LIN {X 0,Y 467.559,Z 348.243,A -85,B 0,C 180,E1 -7440.293,E2 -7440.293} C_VEL
LIN {X 0,Y 467.621,Z 348.236,A -85,B 0,C 180,E1 -7443.199,E2 -7443.199} C_VEL
LIN {X 0,Y 467.597,Z 348.241,A -85,B 0,C 180,E1 -7446.467,E2 -7446.467} C_VEL
LIN {X 0,Y 467.627,Z 348.233,A -85,B 0,C 180,E1 -7449.776,E2 -7449.776} C_VEL
LIN {X 0,Y 467.613,Z 348.24,A -85,B 0,C 180,E1 -7452.506,E2 -7452.506} C_VEL
LIN {X 0,Y 467.61,Z 348.237,A -85,B 0,C 180,E1 -7455.196,E2 -7455.196} C_VEL
LIN {X 0,Y 467.659,Z 348.229,A -85,B 0,C 180,E1 -7457.854,E2 -7457.854} C_VEL
LIN {X 0,Y 467.685,Z 348.227,A -85,B 0,C 180,E1 -7461.356,E2 -7461.356} C_VEL
LIN {X 0,Y 467.738,Z 348.22,A -85,B 0,C 180,E1 -7463.962,E2 -7463.962} C_VEL
LIN {X 0,Y 467.863,Z 348.204,A -85,B 0,C 180,E1 -7467.416,E2 -7467.416} C_VEL
LIN {X 0,Y 467.885,Z 348.203,A -85,B 0,C 180,E1 -7469.999,E2 -7469.999} C_VEL
LIN {X 0,Y 467.862,Z 348.207,A -85,B 0,C 180,E1 -7472.582,E2 -7472.582} C_VEL
LIN {X 0,Y 467.747,Z 348.221,A -85,B 0,C 180,E1 -7476.036,E2 -7476.036} C_VEL
LIN {X 0,Y 467.683,Z 348.229,A -85,B 0,C 180,E1 -7478.642,E2 -7478.642} C_VEL
LIN {X 0,Y 467.656,Z 348.234,A -85,B 0,C 180,E1 -7482.144,E2 -7482.144} C_VEL
LIN {X 0,Y 467.666,Z 348.23,A -85,B 0,C 180,E1 -7485.892,E2 -7485.892} C_VEL
LIN {X 0,Y 467.623,Z 348.233,A -85,B 0,C 180,E1 -7489.307,E2 -7489.307} C_VEL
LIN {X 0,Y 467.534,Z 348.249,A -85,B 0,C 180,E1 -7492.073,E2 -7492.073} C_VEL
LIN {X 0,Y 467.601,Z 348.237,A -85,B 0,C 180,E1 -7494.886,E2 -7494.886} C_VEL
LIN {X 0,Y 467.625,Z 348.235,A -85,B 0,C 180,E1 -7497.767,E2 -7497.767} C_VEL
LIN {X 0,Y 467.569,Z 348.24,A -85,B 0,C 180,E1 -7501.045,E2 -7501.045} C_VEL
LIN {X 0,Y 467.586,Z 348.242,A -85,B 0,C 180,E1 -7504.242,E2 -7504.242} C_VEL
LIN {X 0,Y 467.547,Z 348.242,A -85,B 0,C 180,E1 -7507.186,E2 -7507.186} C_VEL
LIN {X 0,Y 467.596,Z 348.24,A -85,B 0,C 180,E1 -7510.261,E2 -7510.261} C_VEL
LIN {X 0,Y 467.613,Z 348.235,A -85,B 0,C 180,E1 -7512.57,E2 -7512.57} C_VEL
LIN {X 0,Y 467.568,Z 348.243,A -85,B 0,C 180,E1 -7516.175,E2 -7516.175} C_VEL
LIN {X 0,Y 467.584,Z 348.238,A -85,B 0,C 180,E1 -7518.72,E2 -7518.72} C_VEL
LIN {X 0,Y 467.572,Z 348.24,A -85,B 0,C 180,E1 -7521.405,E2 -7521.405} C_VEL
LIN {X 0,Y 467.555,Z 348.243,A -85,B 0,C 180,E1 -7524.259,E2 -7524.259} C_VEL
LIN {X 0,Y 467.574,Z 348.24,A -85,B 0,C 180,E1 -7527.32,E2 -7527.32} C_VEL
LIN {X 0,Y 467.569,Z 348.239,A -85,B 0,C 180,E1 -7530.665,E2 -7530.665} C_VEL
LIN {X 0,Y 467.619,Z 348.234,A -85,B 0,C 180,E1 -7533.2,E2 -7533.2} C_VEL
LIN {X 0,Y 467.583,Z 348.238,A -85,B 0,C 180,E1 -7536.467,E2 -7536.467} C_VEL
LIN {X 0,Y 467.614,Z 348.24,A -85,B 0,C 180,E1 -7539.777,E2 -7539.777} C_VEL
LIN {X 0,Y 467.6,Z 348.235,A -85,B 0,C 180,E1 -7542.506,E2 -7542.506} C_VEL
LIN {X 0,Y 467.597,Z 348.237,A -85,B 0,C 180,E1 -7545.196,E2 -7545.196} C_VEL
LIN {X 0,Y 467.673,Z 348.23,A -85,B 0,C 180,E1 -7547.855,E2 -7547.855} C_VEL
LIN {X 0,Y 467.673,Z 348.23,A -85,B 0,C 180,E1 -7551.357,E2 -7551.357} C_VEL
LIN {X 0,Y 467.734,Z 348.221,A -85,B 0,C 180,E1 -7553.963,E2 -7553.963} C_VEL
LIN {X 0,Y 467.851,Z 348.209,A -85,B 0,C 180,E1 -7557.417,E2 -7557.417} C_VEL
LIN {X 0,Y 467.873,Z 348.202,A -85,B 0,C 180,E1 -7560,E2 -7560} C_VEL
LIN {X 0,Y 467.852,Z 348.203,A -85,B 0,C 180,E1 -7562.583,E2 -7562.583} C_VEL
LIN {X 0,Y 467.742,Z 348.218,A -85,B 0,C 180,E1 -7566.038,E2 -7566.038} C_VEL
LIN {X 0,Y 467.673,Z 348.225,A -85,B 0,C 180,E1 -7568.643,E2 -7568.643} C_VEL
LIN {X 0,Y 467.682,Z 348.224,A -85,B 0,C 180,E1 -7572.379,E2 -7572.379} C_VEL
LIN {X 0,Y 467.64,Z 348.231,A -85,B 0,C 180,E1 -7575.886,E2 -7575.886} C_VEL
LIN {X 0,Y 467.615,Z 348.24,A -85,B 0,C 180,E1 -7579.308,E2 -7579.308} C_VEL
LIN {X 0,Y 467.528,Z 348.244,A -85,B 0,C 180,E1 -7582.074,E2 -7582.074} C_VEL
LIN {X 0,Y 467.595,Z 348.238,A -85,B 0,C 180,E1 -7584.888,E2 -7584.888} C_VEL
LIN {X 0,Y 467.619,Z 348.234,A -85,B 0,C 180,E1 -7587.769,E2 -7587.769} C_VEL
LIN {X 0,Y 467.561,Z 348.245,A -85,B 0,C 180,E1 -7591.046,E2 -7591.046} C_VEL
LIN {X 0,Y 467.582,Z 348.237,A -85,B 0,C 180,E1 -7594.244,E2 -7594.244} C_VEL
LIN {X 0,Y 467.546,Z 348.249,A -85,B 0,C 180,E1 -7597.188,E2 -7597.188} C_VEL
LIN {X 0,Y 467.592,Z 348.236,A -85,B 0,C 180,E1 -7600.263,E2 -7600.263} C_VEL
LIN {X 0,Y 467.613,Z 348.235,A -85,B 0,C 180,E1 -7602.572,E2 -7602.572} C_VEL
LIN {X 0,Y 467.569,Z 348.239,A -85,B 0,C 180,E1 -7606.177,E2 -7606.177} C_VEL
LIN {X 0,Y 467.585,Z 348.24,A -85,B 0,C 180,E1 -7608.723,E2 -7608.723} C_VEL
LIN {X 0,Y 467.575,Z 348.241,A -85,B 0,C 180,E1 -7611.408,E2 -7611.408} C_VEL
LIN {X 0,Y 467.56,Z 348.241,A -85,B 0,C 180,E1 -7614.261,E2 -7614.261} C_VEL
LIN {X 0,Y 467.579,Z 348.241,A -85,B 0,C 180,E1 -7617.322,E2 -7617.322} C_VEL
LIN {X 0,Y 467.577,Z 348.246,A -85,B 0,C 180,E1 -7620.666,E2 -7620.666} C_VEL
LIN {X 0,Y 467.629,Z 348.338,A -85,B 0,C 180,E1 -7621.989,E2 -7621.989} C_VEL
LIN {X 0,Y 470.457,Z 361.803,A -85,B 0,C 180,E1 -7624.329,E2 -7624.329} C_VEL
LIN {X 0,Y 470.48,Z 367.676,A -85,B 0,C 180,E1 -7625.276,E2 -7625.276} C_VEL
LIN {X 0,Y 469.476,Z 388.188,A -85,B 0,C 180,E1 -7628.508,E2 -7628.508} C_VEL
LIN {X 0,Y 468.653,Z 408.371,A -85,B 0,C 180,E1 -7631.645,E2 -7631.645} C_VEL
LIN {X 0,Y 468.38,Z 417.251,A -85,B 0,C 180,E1 -7633.015,E2 -7633.015} C_VEL
LIN {X 0,Y 470.991,Z 437.71,A -85,B 0,C 180,E1 -7633.47,E2 -7633.47} C_VEL
LIN {X 0,Y 470.045,Z 526.671,A -85,B 0,C 180,E1 -7634.999,E2 -7634.999} C_VEL
LIN {X 0,Y 469.641,Z 540.214,A -85,B 0,C 180,E1 -7635.402,E2 -7635.402} C_VEL
LIN {X 0,Y 469.224,Z 553.141,A -85,B 0,C 180,E1 -7635.97,E2 -7635.97} C_VEL
LIN {X 0,Y 468.755,Z 564.967,A -85,B 0,C 180,E1 -7636.674,E2 -7636.674} C_VEL
LIN {X 0,Y 468.309,Z 575.227,A -85,B 0,C 180,E1 -7637.443,E2 -7637.443} C_VEL
LIN {X 0,Y 467.916,Z 585.701,A -85,B 0,C 180,E1 -7638.412,E2 -7638.412} C_VEL
LIN {X 0,Y 467.556,Z 594.368,A -85,B 0,C 180,E1 -7639.39,E2 -7639.39} C_VEL
LIN {X 0,Y 467.25,Z 602.359,A -85,B 0,C 180,E1 -7640.478,E2 -7640.478} C_VEL
LIN {X 0,Y 466.998,Z 610.145,A -85,B 0,C 180,E1 -7641.781,E2 -7641.781} C_VEL
LIN {X 0,Y 466.858,Z 616.396,A -85,B 0,C 180,E1 -7643.084,E2 -7643.084} C_VEL
LIN {X 0,Y 466.797,Z 621.337,A -85,B 0,C 180,E1 -7644.385,E2 -7644.385} C_VEL
LIN {X 0,Y 466.717,Z 625.104,A -85,B 0,C 180,E1 -7645.683,E2 -7645.683} C_VEL
LIN {X 0,Y 466.77,Z 627.045,A -85,B 0,C 180,E1 -7646.548,E2 -7646.548} C_VEL
LIN {X 0,Y 466.778,Z 628.51,A -85,B 0,C 180,E1 -7647.412,E2 -7647.412} C_VEL
LIN {X 0,Y 466.698,Z 629.522,A -85,B 0,C 180,E1 -7648.275,E2 -7648.275} C_VEL
LIN {X 0,Y 466.637,Z 630.128,A -85,B 0,C 180,E1 -7649.138,E2 -7649.138} C_VEL
LIN {X 0,Y 466.631,Z 630.329,A -85,B 0,C 180,E1 -7650.001,E2 -7650.001} C_VEL
LIN {X 0,Y 466.639,Z 630.071,A -85,B 0,C 180,E1 -7650.864,E2 -7650.864} C_VEL
LIN {X 0,Y 466.7,Z 629.4,A -85,B 0,C 180,E1 -7651.727,E2 -7651.727} C_VEL
LIN {X 0,Y 466.8,Z 628.323,A -85,B 0,C 180,E1 -7652.59,E2 -7652.59} C_VEL
LIN {X 0,Y 466.784,Z 625.851,A -85,B 0,C 180,E1 -7653.886,E2 -7653.886} C_VEL
LIN {X 0,Y 466.78,Z 622.335,A -85,B 0,C 180,E1 -7655.184,E2 -7655.184} C_VEL
LIN {X 0,Y 466.88,Z 617.502,A -85,B 0,C 180,E1 -7656.532,E2 -7656.532} C_VEL
LIN {X 0,Y 466.986,Z 610.651,A -85,B 0,C 180,E1 -7658.003,E2 -7658.003} C_VEL
LIN {X 0,Y 467.174,Z 602.973,A -85,B 0,C 180,E1 -7659.308,E2 -7659.308} C_VEL
LIN {X 0,Y 467.499,Z 593.443,A -85,B 0,C 180,E1 -7660.613,E2 -7660.613} C_VEL
LIN {X 0,Y 467.83,Z 583.536,A -85,B 0,C 180,E1 -7661.702,E2 -7661.702} C_VEL
LIN {X 0,Y 468.246,Z 573.369,A -85,B 0,C 180,E1 -7662.615,E2 -7662.615} C_VEL
LIN {X 0,Y 468.759,Z 562.033,A -85,B 0,C 180,E1 -7663.439,E2 -7663.439} C_VEL
LIN {X 0,Y 469.19,Z 549.494,A -85,B 0,C 180,E1 -7664.144,E2 -7664.144} C_VEL
LIN {X 0,Y 469.678,Z 535.736,A -85,B 0,C 180,E1 -7664.71,E2 -7664.71} C_VEL
LIN {X 0,Y 470.109,Z 522.824,A -85,B 0,C 180,E1 -7665.056,E2 -7665.056} C_VEL
LIN {X 0,Y 471.009,Z 436.522,A -85,B 0,C 180,E1 -7666.593,E2 -7666.593} C_VEL
LIN {X 0,Y 468.235,Z 414.349,A -85,B 0,C 180,E1 -7667.146,E2 -7667.146} C_VEL
LIN {X 0,Y 468.975,Z 393.516,A -85,B 0,C 180,E1 -7670.392,E2 -7670.392} C_VEL
LIN {X 0,Y 469.735,Z 376.366,A -85,B 0,C 180,E1 -7673.126,E2 -7673.126} C_VEL
LIN {X 0,Y 470.441,Z 362.283,A -85,B 0,C 180,E1 -7675.437,E2 -7675.437} C_VEL
LIN {X 0,Y 468.39,Z 351.346,A -85,B 0,C 180,E1 -7677.457,E2 -7677.457} C_VEL
LIN {X 0,Y 467.622,Z 348.239,A -85,B 0,C 180,E1 -7678.074,E2 -7678.074} C_VEL
LIN {X 0,Y 467.588,Z 348.242,A -85,B 0,C 180,E1 -7681.741,E2 -7681.741} C_VEL
LIN {X 0,Y 467.571,Z 348.247,A -85,B 0,C 180,E1 -7684.833,E2 -7684.833} C_VEL
LIN {X 0,Y 467.571,Z 348.241,A -85,B 0,C 180,E1 -7688.045,E2 -7688.045} C_VEL
LIN {X 0,Y 467.583,Z 348.243,A -85,B 0,C 180,E1 -7691.277,E2 -7691.277} C_VEL
LIN {X 0,Y 467.559,Z 348.242,A -85,B 0,C 180,E1 -7693.821,E2 -7693.821} C_VEL
LIN {X 0,Y 467.562,Z 348.242,A -85,B 0,C 180,E1 -7696.256,E2 -7696.256} C_VEL
LIN {X 0,Y 467.584,Z 348.242,A -85,B 0,C 180,E1 -7698.723,E2 -7698.723} C_VEL
LIN {X 0,Y 467.57,Z 348.24,A -85,B 0,C 180,E1 -7701.956,E2 -7701.956} C_VEL
LIN {X 0,Y 467.569,Z 348.243,A -85,B 0,C 180,E1 -7705.168,E2 -7705.168} C_VEL
LIN {X 0,Y 467.588,Z 348.239,A -85,B 0,C 180,E1 -7708.26,E2 -7708.26} C_VEL
LIN {X 0,Y 467.582,Z 348.242,A -85,B 0,C 180,E1 -7711.251,E2 -7711.251} C_VEL
LIN {X 0,Y 467.616,Z 348.237,A -85,B 0,C 180,E1 -7714.16,E2 -7714.16} C_VEL
LIN {X 0,Y 467.582,Z 348.245,A -85,B 0,C 180,E1 -7716.996,E2 -7716.996} C_VEL
LIN {X 0,Y 467.628,Z 348.237,A -85,B 0,C 180,E1 -7719.777,E2 -7719.777} C_VEL
LIN {X 0,Y 467.655,Z 348.269,A -85,B 0,C 180,E1 -7721.415,E2 -7721.415} C_VEL
LIN {X 0,Y 468.732,Z 354.118,A -85,B 0,C 180,E1 -7722.999,E2 -7722.999} C_VEL
LIN {X 0,Y 471.442,Z 363.097,A -85,B 0,C 180,E1 -7723.298,E2 -7723.298} C_VEL
LIN {X 0,Y 471.589,Z 367.906,A -85,B 0,C 180,E1 -7723.398,E2 -7723.398} C_VEL
LIN {X 0,Y 470.308,Z 460.031,A -85,B 0,C 180,E1 -7725.09,E2 -7725.09} C_VEL
LIN {X 0,Y 470.102,Z 472.965,A -85,B 0,C 180,E1 -7725.498,E2 -7725.498} C_VEL
LIN {X 0,Y 469.752,Z 484.971,A -85,B 0,C 180,E1 -7726.04,E2 -7726.04} C_VEL
LIN {X 0,Y 469.45,Z 496.77,A -85,B 0,C 180,E1 -7726.758,E2 -7726.758} C_VEL
LIN {X 0,Y 468.982,Z 508.542,A -85,B 0,C 180,E1 -7727.67,E2 -7727.67} C_VEL
LIN {X 0,Y 468.613,Z 517.544,A -85,B 0,C 180,E1 -7728.538,E2 -7728.538} C_VEL
LIN {X 0,Y 468.237,Z 526.749,A -85,B 0,C 180,E1 -7729.623,E2 -7729.623} C_VEL
LIN {X 0,Y 467.818,Z 535.66,A -85,B 0,C 180,E1 -7730.924,E2 -7730.924} C_VEL
LIN {X 0,Y 467.483,Z 542.811,A -85,B 0,C 180,E1 -7732.224,E2 -7732.224} C_VEL
LIN {X 0,Y 467.173,Z 549.054,A -85,B 0,C 180,E1 -7733.679,E2 -7733.679} C_VEL
LIN {X 0,Y 467.075,Z 554.116,A -85,B 0,C 180,E1 -7735.253,E2 -7735.253} C_VEL
LIN {X 0,Y 467.009,Z 557.082,A -85,B 0,C 180,E1 -7736.549,E2 -7736.549} C_VEL
LIN {X 0,Y 466.845,Z 558.521,A -85,B 0,C 180,E1 -7737.411,E2 -7737.411} C_VEL
LIN {X 0,Y 466.667,Z 560.105,A -85,B 0,C 180,E1 -7739.137,E2 -7739.137} C_VEL
LIN {X 0,Y 466.655,Z 560.3,A -85,B 0,C 180,E1 -7740,E2 -7740} C_VEL
LIN {X 0,Y 466.664,Z 560.052,A -85,B 0,C 180,E1 -7740.863,E2 -7740.863} C_VEL
LIN {X 0,Y 466.841,Z 558.333,A -85,B 0,C 180,E1 -7742.588,E2 -7742.588} C_VEL
LIN {X 0,Y 466.975,Z 556.861,A -85,B 0,C 180,E1 -7743.451,E2 -7743.451} C_VEL
LIN {X 0,Y 467.019,Z 553.816,A -85,B 0,C 180,E1 -7744.748,E2 -7744.748} C_VEL
LIN {X 0,Y 467.166,Z 548.664,A -85,B 0,C 180,E1 -7746.318,E2 -7746.318} C_VEL
LIN {X 0,Y 467.356,Z 542.333,A -85,B 0,C 180,E1 -7747.778,E2 -7747.778} C_VEL
LIN {X 0,Y 467.699,Z 535.147,A -85,B 0,C 180,E1 -7749.078,E2 -7749.078} C_VEL
LIN {X 0,Y 468.076,Z 526.163,A -85,B 0,C 180,E1 -7750.38,E2 -7750.38} C_VEL
LIN {X 0,Y 468.481,Z 516.942,A -85,B 0,C 180,E1 -7751.465,E2 -7751.465} C_VEL
LIN {X 0,Y 468.95,Z 506.688,A -85,B 0,C 180,E1 -7752.441,E2 -7752.441} C_VEL
LIN {X 0,Y 469.25,Z 494.356,A -85,B 0,C 180,E1 -7753.379,E2 -7753.379} C_VEL
LIN {X 0,Y 469.629,Z 482.479,A -85,B 0,C 180,E1 -7754.074,E2 -7754.074} C_VEL
LIN {X 0,Y 470.016,Z 469.197,A -85,B 0,C 180,E1 -7754.643,E2 -7754.643} C_VEL
LIN {X 0,Y 470.283,Z 456.11,A -85,B 0,C 180,E1 -7755.022,E2 -7755.022} C_VEL
LIN {X 0,Y 471.084,Z 362.557,A -85,B 0,C 180,E1 -7756.634,E2 -7756.634} C_VEL
LIN {X 0,Y 467.987,Z 350.204,A -85,B 0,C 180,E1 -7756.984,E2 -7756.984} C_VEL
LIN {X 0,Y 467.63,Z 348.238,A -85,B 0,C 180,E1 -7757.492,E2 -7757.492} C_VEL
LIN {X 0,Y 467.627,Z 348.234,A -85,B 0,C 180,E1 -7760.223,E2 -7760.223} C_VEL
LIN {X 0,Y 467.574,Z 348.241,A -85,B 0,C 180,E1 -7763.943,E2 -7763.943} C_VEL
LIN {X 0,Y 467.62,Z 348.237,A -85,B 0,C 180,E1 -7766.8,E2 -7766.8} C_VEL
LIN {X 0,Y 467.559,Z 348.244,A -85,B 0,C 180,E1 -7769.738,E2 -7769.738} C_VEL
LIN {X 0,Y 467.588,Z 348.241,A -85,B 0,C 180,E1 -7772.758,E2 -7772.758} C_VEL
LIN {X 0,Y 467.558,Z 348.243,A -85,B 0,C 180,E1 -7775.889,E2 -7775.889} C_VEL
LIN {X 0,Y 467.587,Z 348.241,A -85,B 0,C 180,E1 -7779.144,E2 -7779.144} C_VEL
LIN {X 0,Y 467.591,Z 348.24,A -85,B 0,C 180,E1 -7782.567,E2 -7782.567} C_VEL
LIN {X 0,Y 467.575,Z 348.243,A -85,B 0,C 180,E1 -7785.053,E2 -7785.053} C_VEL
LIN {X 0,Y 467.593,Z 348.24,A -85,B 0,C 180,E1 -7787.439,E2 -7787.439} C_VEL
LIN {X 0,Y 467.587,Z 348.242,A -85,B 0,C 180,E1 -7790.855,E2 -7790.855} C_VEL
LIN {X 0,Y 467.564,Z 348.242,A -85,B 0,C 180,E1 -7794.26,E2 -7794.26} C_VEL
LIN {X 0,Y 467.586,Z 348.241,A -85,B 0,C 180,E1 -7797.32,E2 -7797.32} C_VEL
LIN {X 0,Y 467.559,Z 348.243,A -85,B 0,C 180,E1 -7800.293,E2 -7800.293} C_VEL
LIN {X 0,Y 466.907,Z 348.327,A -85,B 0,C 180,E1 -7801.013,E2 -7801.013} C_VEL
LIN {X 0,Y 464.063,Z 348.679,A -85,B 0,C 180,E1 -7802.182,E2 -7802.182} C_VEL
LIN {X 0,Y 461.661,Z 348.979,A -85,B 0,C 180,E1 -7803.125,E2 -7803.125} C_VEL
LIN {X 0,Y 460.643,Z 349.104,A -85,B 0,C 180,E1 -7803.854,E2 -7803.854} C_VEL
LIN {X 0,Y 460.568,Z 349.113,A -85,B 0,C 180,E1 -7804.1,E2 -7804.1} C_VEL
LIN {X 0,Y 460.55,Z 349.119,A -85,B 0,C 180,E1 -7806.623,E2 -7806.623} C_VEL
LIN {X 0,Y 460.555,Z 349.115,A -85,B 0,C 180,E1 -7809.452,E2 -7809.452} C_VEL
LIN {X 0,Y 460.563,Z 349.115,A -85,B 0,C 180,E1 -7812.229,E2 -7812.229} C_VEL
LIN {X 0,Y 460.569,Z 349.114,A -85,B 0,C 180,E1 -7814.964,E2 -7814.964} C_VEL
LIN {X 0,Y 460.615,Z 349.111,A -85,B 0,C 180,E1 -7818.558,E2 -7818.558} C_VEL
LIN {X 0,Y 460.698,Z 349.098,A -85,B 0,C 180,E1 -7822.108,E2 -7822.108} C_VEL
LIN {X 0,Y 460.697,Z 349.099,A -85,B 0,C 180,E1 -7824.747,E2 -7824.747} C_VEL
LIN {X 0,Y 460.828,Z 349.08,A -85,B 0,C 180,E1 -7827.377,E2 -7827.377} C_VEL
LIN {X 0,Y 460.856,Z 349.078,A -85,B 0,C 180,E1 -7829.999,E2 -7829.999} C_VEL
LIN {X 0,Y 460.827,Z 349.083,A -85,B 0,C 180,E1 -7832.621,E2 -7832.621} C_VEL
LIN {X 0,Y 460.713,Z 349.098,A -85,B 0,C 180,E1 -7836.129,E2 -7836.129} C_VEL
LIN {X 0,Y 460.63,Z 349.106,A -85,B 0,C 180,E1 -7838.775,E2 -7838.775} C_VEL
LIN {X 0,Y 460.613,Z 349.11,A -85,B 0,C 180,E1 -7842.444,E2 -7842.444} C_VEL
LIN {X 0,Y 460.621,Z 349.109,A -85,B 0,C 180,E1 -7846.006,E2 -7846.006} C_VEL
LIN {X 0,Y 460.568,Z 349.113,A -85,B 0,C 180,E1 -7849.614,E2 -7849.614} C_VEL
LIN {X 0,Y 460.51,Z 349.122,A -85,B 0,C 180,E1 -7852.427,E2 -7852.427} C_VEL
LIN {X 0,Y 460.566,Z 349.115,A -85,B 0,C 180,E1 -7855.801,E2 -7855.801} C_VEL
LIN {X 0,Y 460.556,Z 349.118,A -85,B 0,C 180,E1 -7858.231,E2 -7858.231} C_VEL
LIN {X 0,Y 460.521,Z 349.118,A -85,B 0,C 180,E1 -7861.283,E2 -7861.283} C_VEL
LIN {X 0,Y 460.53,Z 349.118,A -85,B 0,C 180,E1 -7864.505,E2 -7864.505} C_VEL
LIN {X 0,Y 460.526,Z 349.119,A -85,B 0,C 180,E1 -7867.619,E2 -7867.619} C_VEL
LIN {X 0,Y 460.558,Z 349.116,A -85,B 0,C 180,E1 -7870.272,E2 -7870.272} C_VEL
LIN {X 0,Y 460.518,Z 349.119,A -85,B 0,C 180,E1 -7873.371,E2 -7873.371} C_VEL
LIN {X 0,Y 460.518,Z 349.119,A -85,B 0,C 180,E1 -7876.627,E2 -7876.627} C_VEL
LIN {X 0,Y 460.557,Z 349.118,A -85,B 0,C 180,E1 -7879.726,E2 -7879.726} C_VEL
LIN {X 0,Y 460.521,Z 349.118,A -85,B 0,C 180,E1 -7882.518,E2 -7882.518} C_VEL
LIN {X 0,Y 460.541,Z 349.119,A -85,B 0,C 180,E1 -7885.623,E2 -7885.623} C_VEL
LIN {X 0,Y 460.528,Z 349.116,A -85,B 0,C 180,E1 -7888.744,E2 -7888.744} C_VEL
LIN {X 0,Y 460.55,Z 349.121,A -85,B 0,C 180,E1 -7891.767,E2 -7891.767} C_VEL
LIN {X 0,Y 460.55,Z 349.113,A -85,B 0,C 180,E1 -7894.705,E2 -7894.705} C_VEL
LIN {X 0,Y 460.503,Z 349.124,A -85,B 0,C 180,E1 -7897.571,E2 -7897.571} C_VEL
LIN {X 0,Y 460.56,Z 349.113,A -85,B 0,C 180,E1 -7900.384,E2 -7900.384} C_VEL
LIN {X 0,Y 460.621,Z 349.107,A -85,B 0,C 180,E1 -7904.06,E2 -7904.06} C_VEL
LIN {X 0,Y 460.62,Z 349.111,A -85,B 0,C 180,E1 -7907.666,E2 -7907.666} C_VEL
LIN {X 0,Y 460.62,Z 349.107,A -85,B 0,C 180,E1 -7911.224,E2 -7911.224} C_VEL
LIN {X 0,Y 460.7,Z 349.098,A -85,B 0,C 180,E1 -7913.87,E2 -7913.87} C_VEL
LIN {X 0,Y 460.816,Z 349.085,A -85,B 0,C 180,E1 -7917.378,E2 -7917.378} C_VEL
LIN {X 0,Y 460.844,Z 349.078,A -85,B 0,C 180,E1 -7920,E2 -7920} C_VEL
LIN {X 0,Y 460.817,Z 349.079,A -85,B 0,C 180,E1 -7922.623,E2 -7922.623} C_VEL
LIN {X 0,Y 460.707,Z 349.094,A -85,B 0,C 180,E1 -7926.13,E2 -7926.13} C_VEL
LIN {X 0,Y 460.62,Z 349.105,A -85,B 0,C 180,E1 -7928.776,E2 -7928.776} C_VEL
LIN {X 0,Y 460.624,Z 349.103,A -85,B 0,C 180,E1 -7932.457,E2 -7932.457} C_VEL
LIN {X 0,Y 460.59,Z 349.109,A -85,B 0,C 180,E1 -7935.998,E2 -7935.998} C_VEL
LIN {X 0,Y 460.562,Z 349.114,A -85,B 0,C 180,E1 -7938.903,E2 -7938.903} C_VEL
LIN {X 0,Y 460.507,Z 349.124,A -85,B 0,C 180,E1 -7941.486,E2 -7941.486} C_VEL
LIN {X 0,Y 460.534,Z 349.115,A -85,B 0,C 180,E1 -7944.333,E2 -7944.333} C_VEL
LIN {X 0,Y 460.576,Z 349.117,A -85,B 0,C 180,E1 -7947.244,E2 -7947.244} C_VEL
LIN {X 0,Y 460.503,Z 349.119,A -85,B 0,C 180,E1 -7950.241,E2 -7950.241} C_VEL
LIN {X 0,Y 460.522,Z 349.122,A -85,B 0,C 180,E1 -7953.326,E2 -7953.326} C_VEL
LIN {X 0,Y 460.473,Z 349.124,A -85,B 0,C 180,E1 -7956.53,E2 -7956.53} C_VEL
LIN {X 0,Y 460.572,Z 349.111,A -85,B 0,C 180,E1 -7959.858,E2 -7959.858} C_VEL
LIN {X 0,Y 460.537,Z 349.119,A -85,B 0,C 180,E1 -7962.905,E2 -7962.905} C_VEL
LIN {X 0,Y 460.519,Z 349.118,A -85,B 0,C 180,E1 -7965.83,E2 -7965.83} C_VEL
LIN {X 0,Y 460.538,Z 349.121,A -85,B 0,C 180,E1 -7968.991,E2 -7968.991} C_VEL
LIN {X 0,Y 460.544,Z 349.118,A -85,B 0,C 180,E1 -7971.27,E2 -7971.27} C_VEL
LIN {X 0,Y 460.511,Z 349.121,A -85,B 0,C 180,E1 -7974.556,E2 -7974.556} C_VEL
LIN {X 0,Y 460.531,Z 349.116,A -85,B 0,C 180,E1 -7977.717,E2 -7977.717} C_VEL
LIN {X 0,Y 460.547,Z 349.122,A -85,B 0,C 180,E1 -7980.771,E2 -7980.771} C_VEL
LIN {X 0,Y 460.615,Z 349.21,A -85,B 0,C 180,E1 -7981.773,E2 -7981.773} C_VEL
LIN {X 0,Y 463.432,Z 362.681,A -85,B 0,C 180,E1 -7984.153,E2 -7984.153} C_VEL
LIN {X 0,Y 463.587,Z 367.101,A -85,B 0,C 180,E1 -7984.883,E2 -7984.883} C_VEL
LIN {X 0,Y 462.657,Z 386.732,A -85,B 0,C 180,E1 -7988.027,E2 -7988.027} C_VEL
LIN {X 0,Y 461.713,Z 407.823,A -85,B 0,C 180,E1 -7991.359,E2 -7991.359} C_VEL
LIN {X 0,Y 461.379,Z 416.811,A -85,B 0,C 180,E1 -7992.767,E2 -7992.767} C_VEL
LIN {X 0,Y 464.125,Z 438.104,A -85,B 0,C 180,E1 -7993.252,E2 -7993.252} C_VEL
LIN {X 0,Y 463.091,Z 527.005,A -85,B 0,C 180,E1 -7994.825,E2 -7994.825} C_VEL
LIN {X 0,Y 462.662,Z 541.001,A -85,B 0,C 180,E1 -7995.261,E2 -7995.261} C_VEL
LIN {X 0,Y 462.254,Z 553.006,A -85,B 0,C 180,E1 -7995.81,E2 -7995.81} C_VEL
LIN {X 0,Y 461.726,Z 565.552,A -85,B 0,C 180,E1 -7996.579,E2 -7996.579} C_VEL
LIN {X 0,Y 461.276,Z 575.501,A -85,B 0,C 180,E1 -7997.35,E2 -7997.35} C_VEL
LIN {X 0,Y 460.852,Z 585.942,A -85,B 0,C 180,E1 -7998.344,E2 -7998.344} C_VEL
LIN {X 0,Y 460.44,Z 595.313,A -85,B 0,C 180,E1 -7999.447,E2 -7999.447} C_VEL
LIN {X 0,Y 460.096,Z 604.431,A -85,B 0,C 180,E1 -8000.772,E2 -8000.772} C_VEL
LIN {X 0,Y 459.87,Z 611.757,A -85,B 0,C 180,E1 -8002.095,E2 -8002.095} C_VEL
LIN {X 0,Y 459.771,Z 617.911,A -85,B 0,C 180,E1 -8003.507,E2 -8003.507} C_VEL
LIN {X 0,Y 459.71,Z 622.137,A -85,B 0,C 180,E1 -8004.738,E2 -8004.738} C_VEL
LIN {X 0,Y 459.625,Z 624.526,A -85,B 0,C 180,E1 -8005.616,E2 -8005.616} C_VEL
LIN {X 0,Y 459.699,Z 626.48,A -85,B 0,C 180,E1 -8006.495,E2 -8006.495} C_VEL
LIN {X 0,Y 459.692,Z 627.96,A -85,B 0,C 180,E1 -8007.372,E2 -8007.372} C_VEL
LIN {X 0,Y 459.637,Z 628.98,A -85,B 0,C 180,E1 -8008.249,E2 -8008.249} C_VEL
LIN {X 0,Y 459.569,Z 629.59,A -85,B 0,C 180,E1 -8009.125,E2 -8009.125} C_VEL
LIN {X 0,Y 459.56,Z 629.793,A -85,B 0,C 180,E1 -8010.001,E2 -8010.001} C_VEL
LIN {X 0,Y 459.571,Z 629.539,A -85,B 0,C 180,E1 -8010.877,E2 -8010.877} C_VEL
LIN {X 0,Y 459.639,Z 628.864,A -85,B 0,C 180,E1 -8011.753,E2 -8011.753} C_VEL
LIN {X 0,Y 459.714,Z 627.779,A -85,B 0,C 180,E1 -8012.63,E2 -8012.63} C_VEL
LIN {X 0,Y 459.695,Z 625.298,A -85,B 0,C 180,E1 -8013.946,E2 -8013.946} C_VEL
LIN {X 0,Y 459.714,Z 621.774,A -85,B 0,C 180,E1 -8015.264,E2 -8015.264} C_VEL
LIN {X 0,Y 459.803,Z 616.344,A -85,B 0,C 180,E1 -8016.778,E2 -8016.778} C_VEL
LIN {X 0,Y 459.911,Z 610.058,A -85,B 0,C 180,E1 -8018.127,E2 -8018.127} C_VEL
LIN {X 0,Y 460.12,Z 602.352,A -85,B 0,C 180,E1 -8019.452,E2 -8019.452} C_VEL
LIN {X 0,Y 460.467,Z 592.806,A -85,B 0,C 180,E1 -8020.777,E2 -8020.777} C_VEL
LIN {X 0,Y 460.852,Z 582.893,A -85,B 0,C 180,E1 -8021.882,E2 -8021.882} C_VEL
LIN {X 0,Y 461.298,Z 571.547,A -85,B 0,C 180,E1 -8022.907,E2 -8022.907} C_VEL
LIN {X 0,Y 461.875,Z 559.623,A -85,B 0,C 180,E1 -8023.755,E2 -8023.755} C_VEL
LIN {X 0,Y 462.404,Z 546.596,A -85,B 0,C 180,E1 -8024.468,E2 -8024.468} C_VEL
LIN {X 0,Y 462.861,Z 533.515,A -85,B 0,C 180,E1 -8024.988,E2 -8024.988} C_VEL
LIN {X 0,Y 463.297,Z 519.68,A -85,B 0,C 180,E1 -8025.339,E2 -8025.339} C_VEL
LIN {X 0,Y 464.308,Z 437.682,A -85,B 0,C 180,E1 -8026.84,E2 -8026.84} C_VEL
LIN {X 0,Y 461.277,Z 414.138,A -85,B 0,C 180,E1 -8027.441,E2 -8027.441} C_VEL
LIN {X 0,Y 461.24,Z 413.249,A -85,B 0,C 180,E1 -8027.524,E2 -8027.524} C_VEL
LIN {X 0,Y 462.007,Z 394.637,A -85,B 0,C 180,E1 -8030.48,E2 -8030.48} C_VEL
LIN {X 0,Y 462.878,Z 376.201,A -85,B 0,C 180,E1 -8033.489,E2 -8033.489} C_VEL
LIN {X 0,Y 463.607,Z 365.038,A -85,B 0,C 180,E1 -8035.358,E2 -8035.358} C_VEL
LIN {X 0,Y 462.855,Z 359.427,A -85,B 0,C 180,E1 -8036.381,E2 -8036.381} C_VEL
LIN {X 0,Y 460.579,Z 349.116,A -85,B 0,C 180,E1 -8038.418,E2 -8038.418} C_VEL
LIN {X 0,Y 460.526,Z 349.123,A -85,B 0,C 180,E1 -8041.284,E2 -8041.284} C_VEL
LIN {X 0,Y 460.538,Z 349.12,A -85,B 0,C 180,E1 -8044.506,E2 -8044.506} C_VEL
LIN {X 0,Y 460.507,Z 349.123,A -85,B 0,C 180,E1 -8047.624,E2 -8047.624} C_VEL
LIN {X 0,Y 460.547,Z 349.117,A -85,B 0,C 180,E1 -8050.27,E2 -8050.27} C_VEL
LIN {X 0,Y 460.506,Z 349.123,A -85,B 0,C 180,E1 -8053.376,E2 -8053.376} C_VEL
LIN {X 0,Y 460.506,Z 349.123,A -85,B 0,C 180,E1 -8056.625,E2 -8056.625} C_VEL
LIN {X 0,Y 460.547,Z 349.116,A -85,B 0,C 180,E1 -8059.731,E2 -8059.731} C_VEL
LIN {X 0,Y 460.505,Z 349.123,A -85,B 0,C 180,E1 -8062.524,E2 -8062.524} C_VEL
LIN {X 0,Y 460.551,Z 349.115,A -85,B 0,C 180,E1 -8065.624,E2 -8065.624} C_VEL
LIN {X 0,Y 460.543,Z 349.12,A -85,B 0,C 180,E1 -8068.745,E2 -8068.745} C_VEL
LIN {X 0,Y 460.587,Z 349.112,A -85,B 0,C 180,E1 -8072.254,E2 -8072.254} C_VEL
LIN {X 0,Y 460.564,Z 349.119,A -85,B 0,C 180,E1 -8074.706,E2 -8074.706} C_VEL
LIN {X 0,Y 460.516,Z 349.122,A -85,B 0,C 180,E1 -8077.571,E2 -8077.571} C_VEL
LIN {X 0,Y 460.58,Z 349.117,A -85,B 0,C 180,E1 -8080.8,E2 -8080.8} C_VEL
LIN {X 0,Y 460.596,Z 349.172,A -85,B 0,C 180,E1 -8081.091,E2 -8081.091} C_VEL
LIN {X 0,Y 461.661,Z 354.639,A -85,B 0,C 180,E1 -8082.66,E2 -8082.66} C_VEL
LIN {X 0,Y 464.627,Z 363.647,A -85,B 0,C 180,E1 -8082.998,E2 -8082.998} C_VEL
LIN {X 0,Y 464.969,Z 366.827,A -85,B 0,C 180,E1 -8083.079,E2 -8083.079} C_VEL
LIN {X 0,Y 463.503,Z 460.986,A -85,B 0,C 180,E1 -8084.865,E2 -8084.865} C_VEL
LIN {X 0,Y 463.269,Z 473.746,A -85,B 0,C 180,E1 -8085.279,E2 -8085.279} C_VEL
LIN {X 0,Y 462.915,Z 485.677,A -85,B 0,C 180,E1 -8085.829,E2 -8085.829} C_VEL
LIN {X 0,Y 462.569,Z 497.774,A -85,B 0,C 180,E1 -8086.58,E2 -8086.58} C_VEL
LIN {X 0,Y 462.078,Z 509.188,A -85,B 0,C 180,E1 -8087.482,E2 -8087.482} C_VEL
LIN {X 0,Y 461.684,Z 518.172,A -85,B 0,C 180,E1 -8088.364,E2 -8088.364} C_VEL
LIN {X 0,Y 461.282,Z 527.364,A -85,B 0,C 180,E1 -8089.465,E2 -8089.465} C_VEL
LIN {X 0,Y 460.839,Z 536.277,A -85,B 0,C 180,E1 -8090.785,E2 -8090.785} C_VEL
LIN {X 0,Y 460.495,Z 543.421,A -85,B 0,C 180,E1 -8092.105,E2 -8092.105} C_VEL
LIN {X 0,Y 460.194,Z 548.853,A -85,B 0,C 180,E1 -8093.363,E2 -8093.363} C_VEL
LIN {X 0,Y 460.125,Z 553.474,A -85,B 0,C 180,E1 -8094.742,E2 -8094.742} C_VEL
LIN {X 0,Y 459.979,Z 555.791,A -85,B 0,C 180,E1 -8095.619,E2 -8095.619} C_VEL
LIN {X 0,Y 459.963,Z 557.662,A -85,B 0,C 180,E1 -8096.496,E2 -8096.496} C_VEL
LIN {X 0,Y 459.794,Z 559.093,A -85,B 0,C 180,E1 -8097.372,E2 -8097.372} C_VEL
LIN {X 0,Y 459.659,Z 560.079,A -85,B 0,C 180,E1 -8098.248,E2 -8098.248} C_VEL
LIN {X 0,Y 459.598,Z 560.663,A -85,B 0,C 180,E1 -8099.124,E2 -8099.124} C_VEL
LIN {X 0,Y 459.583,Z 560.846,A -85,B 0,C 180,E1 -8100,E2 -8100} C_VEL
LIN {X 0,Y 459.595,Z 560.58,A -85,B 0,C 180,E1 -8100.876,E2 -8100.876} C_VEL
LIN {X 0,Y 459.789,Z 558.828,A -85,B 0,C 180,E1 -8102.628,E2 -8102.628} C_VEL
LIN {X 0,Y 459.899,Z 557.333,A -85,B 0,C 180,E1 -8103.504,E2 -8103.504} C_VEL
LIN {X 0,Y 459.966,Z 554.253,A -85,B 0,C 180,E1 -8104.821,E2 -8104.821} C_VEL
LIN {X 0,Y 460.057,Z 550.095,A -85,B 0,C 180,E1 -8106.139,E2 -8106.139} C_VEL
LIN {X 0,Y 460.27,Z 543.702,A -85,B 0,C 180,E1 -8107.678,E2 -8107.678} C_VEL
LIN {X 0,Y 460.612,Z 536.731,A -85,B 0,C 180,E1 -8108.998,E2 -8108.998} C_VEL
LIN {X 0,Y 460.937,Z 529.608,A -85,B 0,C 180,E1 -8110.099,E2 -8110.099} C_VEL
LIN {X 0,Y 461.303,Z 521.002,A -85,B 0,C 180,E1 -8111.201,E2 -8111.201} C_VEL
LIN {X 0,Y 461.809,Z 510.349,A -85,B 0,C 180,E1 -8112.302,E2 -8112.302} C_VEL
LIN {X 0,Y 462.19,Z 499.795,A -85,B 0,C 180,E1 -8113.184,E2 -8113.184} C_VEL
LIN {X 0,Y 462.568,Z 488.173,A -85,B 0,C 180,E1 -8113.957,E2 -8113.957} C_VEL
LIN {X 0,Y 462.944,Z 476.17,A -85,B 0,C 180,E1 -8114.563,E2 -8114.563} C_VEL
LIN {X 0,Y 463.216,Z 462.439,A -85,B 0,C 180,E1 -8115.06,E2 -8115.06} C_VEL
LIN {X 0,Y 463.402,Z 448.461,A -85,B 0,C 180,E1 -8115.363,E2 -8115.363} C_VEL
LIN {X 0,Y 464.387,Z 364.701,A -85,B 0,C 180,E1 -8116.825,E2 -8116.825} C_VEL
LIN {X 0,Y 461.858,Z 354.086,A -85,B 0,C 180,E1 -8117.109,E2 -8117.109} C_VEL
LIN {X 0,Y 460.859,Z 350.615,A -85,B 0,C 180,E1 -8117.235,E2 -8117.235} C_VEL
LIN {X 0,Y 460.6,Z 349.113,A -85,B 0,C 180,E1 -8117.654,E2 -8117.654} C_VEL
LIN {X 0,Y 460.556,Z 349.115,A -85,B 0,C 180,E1 -8120.547,E2 -8120.547} C_VEL
LIN {X 0,Y 460.539,Z 349.119,A -85,B 0,C 180,E1 -8123.704,E2 -8123.704} C_VEL
LIN {X 0,Y 460.563,Z 349.114,A -85,B 0,C 180,E1 -8126.265,E2 -8126.265} C_VEL
LIN {X 0,Y 460.545,Z 349.118,A -85,B 0,C 180,E1 -8129.231,E2 -8129.231} C_VEL
LIN {X 0,Y 460.536,Z 349.117,A -85,B 0,C 180,E1 -8132.284,E2 -8132.284} C_VEL
LIN {X 0,Y 460.515,Z 349.122,A -85,B 0,C 180,E1 -8135.445,E2 -8135.445} C_VEL
LIN {X 0,Y 460.549,Z 349.119,A -85,B 0,C 180,E1 -8138.897,E2 -8138.897} C_VEL
LIN {X 0,Y 460.527,Z 349.118,A -85,B 0,C 180,E1 -8142.181,E2 -8142.181} C_VEL
LIN {X 0,Y 460.521,Z 349.121,A -85,B 0,C 180,E1 -8145.411,E2 -8145.411} C_VEL
LIN {X 0,Y 460.536,Z 349.118,A -85,B 0,C 180,E1 -8148.397,E2 -8148.397} C_VEL
LIN {X 0,Y 460.531,Z 349.12,A -85,B 0,C 180,E1 -8151.266,E2 -8151.266} C_VEL
LIN {X 0,Y 460.515,Z 349.123,A -85,B 0,C 180,E1 -8154.554,E2 -8154.554} C_VEL
LIN {X 0,Y 460.535,Z 349.117,A -85,B 0,C 180,E1 -8157.715,E2 -8157.715} C_VEL
LIN {X 0,Y 460.544,Z 349.119,A -85,B 0,C 180,E1 -8160.768,E2 -8160.768} C_VEL
LIN {X 0,Y 460.567,Z 349.113,A -85,B 0,C 180,E1 -8163.734,E2 -8163.734} C_VEL
LIN {X 0,Y 460.568,Z 349.113,A -85,B 0,C 180,E1 -8164.1,E2 -8164.1} C_VEL
LIN {X 0,Y 459.912,Z 349.198,A -85,B 0,C 180,E1 -8164.83,E2 -8164.83} C_VEL
LIN {X 0,Y 457.023,Z 349.556,A -85,B 0,C 180,E1 -8166.014,E2 -8166.014} C_VEL
LIN {X 0,Y 454.579,Z 349.861,A -85,B 0,C 180,E1 -8166.969,E2 -8166.969} C_VEL
LIN {X 0,Y 453.545,Z 349.988,A -85,B 0,C 180,E1 -8167.708,E2 -8167.708} C_VEL
LIN {X 0,Y 453.47,Z 349.997,A -85,B 0,C 180,E1 -8167.958,E2 -8167.958} C_VEL
LIN {X 0,Y 453.526,Z 349.992,A -85,B 0,C 180,E1 -8171.008,E2 -8171.008} C_VEL
LIN {X 0,Y 453.572,Z 349.984,A -85,B 0,C 180,E1 -8173.879,E2 -8173.879} C_VEL
LIN {X 0,Y 453.566,Z 349.985,A -85,B 0,C 180,E1 -8177.47,E2 -8177.47} C_VEL
LIN {X 0,Y 453.595,Z 349.983,A -85,B 0,C 180,E1 -8181.086,E2 -8181.086} C_VEL
LIN {X 0,Y 453.672,Z 349.972,A -85,B 0,C 180,E1 -8183.774,E2 -8183.774} C_VEL
LIN {X 0,Y 453.768,Z 349.96,A -85,B 0,C 180,E1 -8187.336,E2 -8187.336} C_VEL
LIN {X 0,Y 453.826,Z 349.954,A -85,B 0,C 180,E1 -8189.999,E2 -8189.999} C_VEL
LIN {X 0,Y 453.767,Z 349.962,A -85,B 0,C 180,E1 -8192.662,E2 -8192.662} C_VEL
LIN {X 0,Y 453.68,Z 349.975,A -85,B 0,C 180,E1 -8196.224,E2 -8196.224} C_VEL
LIN {X 0,Y 453.593,Z 349.983,A -85,B 0,C 180,E1 -8198.912,E2 -8198.912} C_VEL
LIN {X 0,Y 453.563,Z 349.988,A -85,B 0,C 180,E1 -8202.528,E2 -8202.528} C_VEL
LIN {X 0,Y 453.556,Z 349.991,A -85,B 0,C 180,E1 -8206.194,E2 -8206.194} C_VEL
LIN {X 0,Y 453.519,Z 349.991,A -85,B 0,C 180,E1 -8209.04,E2 -8209.04} C_VEL
LIN {X 0,Y 453.475,Z 349.998,A -85,B 0,C 180,E1 -8211.835,E2 -8211.835} C_VEL
LIN {X 0,Y 453.512,Z 349.992,A -85,B 0,C 180,E1 -8214.733,E2 -8214.733} C_VEL
LIN {X 0,Y 453.536,Z 349.993,A -85,B 0,C 180,E1 -8217.96,E2 -8217.96} C_VEL
LIN {X 0,Y 453.48,Z 349.996,A -85,B 0,C 180,E1 -8220.758,E2 -8220.758} C_VEL
LIN {X 0,Y 453.474,Z 350,A -85,B 0,C 180,E1 -8223.911,E2 -8223.911} C_VEL
LIN {X 0,Y 453.467,Z 349.996,A -85,B 0,C 180,E1 -8227.187,E2 -8227.187} C_VEL
LIN {X 0,Y 453.531,Z 349.989,A -85,B 0,C 180,E1 -8229.444,E2 -8229.444} C_VEL
LIN {X 0,Y 453.485,Z 349.994,A -85,B 0,C 180,E1 -8232.99,E2 -8232.99} C_VEL
LIN {X 0,Y 453.47,Z 350.001,A -85,B 0,C 180,E1 -8235.78,E2 -8235.78} C_VEL
LIN {X 0,Y 453.49,Z 349.996,A -85,B 0,C 180,E1 -8238.211,E2 -8238.211} C_VEL
LIN {X 0,Y 453.528,Z 349.989,A -85,B 0,C 180,E1 -8240.786,E2 -8240.786} C_VEL
LIN {X 0,Y 453.45,Z 350.004,A -85,B 0,C 180,E1 -8243.917,E2 -8243.917} C_VEL
LIN {X 0,Y 453.475,Z 349.995,A -85,B 0,C 180,E1 -8247.151,E2 -8247.151} C_VEL
LIN {X 0,Y 453.505,Z 349.993,A -85,B 0,C 180,E1 -8250.271,E2 -8250.271} C_VEL
LIN {X 0,Y 453.505,Z 349.993,A -85,B 0,C 180,E1 -8253.294,E2 -8253.294} C_VEL
LIN {X 0,Y 453.494,Z 349.994,A -85,B 0,C 180,E1 -8256.238,E2 -8256.238} C_VEL
LIN {X 0,Y 453.473,Z 349.996,A -85,B 0,C 180,E1 -8259.117,E2 -8259.117} C_VEL
LIN {X 0,Y 453.503,Z 349.995,A -85,B 0,C 180,E1 -8261.944,E2 -8261.944} C_VEL
LIN {X 0,Y 453.54,Z 349.986,A -85,B 0,C 180,E1 -8264.726,E2 -8264.726} C_VEL
LIN {X 0,Y 453.592,Z 349.985,A -85,B 0,C 180,E1 -8267.472,E2 -8267.472} C_VEL
LIN {X 0,Y 453.584,Z 349.982,A -85,B 0,C 180,E1 -8271.087,E2 -8271.087} C_VEL
LIN {X 0,Y 453.668,Z 349.975,A -85,B 0,C 180,E1 -8273.775,E2 -8273.775} C_VEL
LIN {X 0,Y 453.757,Z 349.964,A -85,B 0,C 180,E1 -8277.337,E2 -8277.337} C_VEL
LIN {X 0,Y 453.815,Z 349.954,A -85,B 0,C 180,E1 -8280,E2 -8280} C_VEL
LIN {X 0,Y 453.757,Z 349.959,A -85,B 0,C 180,E1 -8282.663,E2 -8282.663} C_VEL
LIN {X 0,Y 453.673,Z 349.969,A -85,B 0,C 180,E1 -8286.225,E2 -8286.225} C_VEL
LIN {X 0,Y 453.584,Z 349.982,A -85,B 0,C 180,E1 -8288.914,E2 -8288.914} C_VEL
LIN {X 0,Y 453.592,Z 349.979,A -85,B 0,C 180,E1 -8292.551,E2 -8292.551} C_VEL
LIN {X 0,Y 453.535,Z 349.987,A -85,B 0,C 180,E1 -8296.196,E2 -8296.196} C_VEL
LIN {X 0,Y 453.512,Z 349.993,A -85,B 0,C 180,E1 -8299.042,E2 -8299.042} C_VEL
LIN {X 0,Y 453.468,Z 349.997,A -85,B 0,C 180,E1 -8301.837,E2 -8301.837} C_VEL
LIN {X 0,Y 453.506,Z 349.992,A -85,B 0,C 180,E1 -8304.735,E2 -8304.735} C_VEL
LIN {X 0,Y 453.529,Z 349.988,A -85,B 0,C 180,E1 -8307.962,E2 -8307.962} C_VEL
LIN {X 0,Y 453.459,Z 350,A -85,B 0,C 180,E1 -8311.526,E2 -8311.526} C_VEL
LIN {X 0,Y 453.482,Z 349.996,A -85,B 0,C 180,E1 -8314.779,E2 -8314.779} C_VEL
LIN {X 0,Y 453.479,Z 349.995,A -85,B 0,C 180,E1 -8318.31,E2 -8318.31} C_VEL
LIN {X 0,Y 453.51,Z 349.992,A -85,B 0,C 180,E1 -8320.607,E2 -8320.607} C_VEL
LIN {X 0,Y 453.477,Z 350,A -85,B 0,C 180,E1 -8323.249,E2 -8323.249} C_VEL
LIN {X 0,Y 453.472,Z 349.996,A -85,B 0,C 180,E1 -8325.782,E2 -8325.782} C_VEL
LIN {X 0,Y 453.491,Z 349.993,A -85,B 0,C 180,E1 -8328.212,E2 -8328.212} C_VEL
LIN {X 0,Y 453.529,Z 349.992,A -85,B 0,C 180,E1 -8330.788,E2 -8330.788} C_VEL
LIN {X 0,Y 453.455,Z 349.998,A -85,B 0,C 180,E1 -8333.919,E2 -8333.919} C_VEL
LIN {X 0,Y 453.48,Z 349.999,A -85,B 0,C 180,E1 -8337.153,E2 -8337.153} C_VEL
LIN {X 0,Y 453.512,Z 349.996,A -85,B 0,C 180,E1 -8340.272,E2 -8340.272} C_VEL
LIN {X 0,Y 453.544,Z 350.061,A -85,B 0,C 180,E1 -8341.552,E2 -8341.552} C_VEL
LIN {X 0,Y 456.643,Z 365.044,A -85,B 0,C 180,E1 -8344.23,E2 -8344.23} C_VEL
LIN {X 0,Y 456.222,Z 376.727,A -85,B 0,C 180,E1 -8346.149,E2 -8346.149} C_VEL
LIN {X 0,Y 455.258,Z 395.633,A -85,B 0,C 180,E1 -8349.204,E2 -8349.204} C_VEL
LIN {X 0,Y 454.384,Z 416.316,A -85,B 0,C 180,E1 -8352.505,E2 -8352.505} C_VEL
LIN {X 0,Y 457.254,Z 439.43,A -85,B 0,C 180,E1 -8353.053,E2 -8353.053} C_VEL
LIN {X 0,Y 456.197,Z 525.959,A -85,B 0,C 180,E1 -8354.618,E2 -8354.618} C_VEL
LIN {X 0,Y 455.74,Z 540.088,A -85,B 0,C 180,E1 -8355.06,E2 -8355.06} C_VEL
LIN {X 0,Y 455.266,Z 552.713,A -85,B 0,C 180,E1 -8355.644,E2 -8355.644} C_VEL
LIN {X 0,Y 454.765,Z 564.42,A -85,B 0,C 180,E1 -8356.37,E2 -8356.37} C_VEL
LIN {X 0,Y 454.243,Z 575.685,A -85,B 0,C 180,E1 -8357.255,E2 -8357.255} C_VEL
LIN {X 0,Y 453.771,Z 586.068,A -85,B 0,C 180,E1 -8358.272,E2 -8358.272} C_VEL
LIN {X 0,Y 453.309,Z 596.165,A -85,B 0,C 180,E1 -8359.505,E2 -8359.505} C_VEL
LIN {X 0,Y 453.001,Z 605.055,A -85,B 0,C 180,E1 -8360.851,E2 -8360.851} C_VEL
LIN {X 0,Y 452.76,Z 612.121,A -85,B 0,C 180,E1 -8362.195,E2 -8362.195} C_VEL
LIN {X 0,Y 452.632,Z 618.596,A -85,B 0,C 180,E1 -8363.761,E2 -8363.761} C_VEL
LIN {X 0,Y 452.571,Z 622.803,A -85,B 0,C 180,E1 -8365.101,E2 -8365.101} C_VEL
LIN {X 0,Y 452.63,Z 625.904,A -85,B 0,C 180,E1 -8366.44,E2 -8366.44} C_VEL
LIN {X 0,Y 452.611,Z 627.402,A -85,B 0,C 180,E1 -8367.331,E2 -8367.331} C_VEL
LIN {X 0,Y 452.577,Z 628.432,A -85,B 0,C 180,E1 -8368.221,E2 -8368.221} C_VEL
LIN {X 0,Y 452.504,Z 629.046,A -85,B 0,C 180,E1 -8369.111,E2 -8369.111} C_VEL
LIN {X 0,Y 452.492,Z 629.254,A -85,B 0,C 180,E1 -8370.001,E2 -8370.001} C_VEL
LIN {X 0,Y 452.506,Z 629.007,A -85,B 0,C 180,E1 -8370.891,E2 -8370.891} C_VEL
LIN {X 0,Y 452.579,Z 628.333,A -85,B 0,C 180,E1 -8371.781,E2 -8371.781} C_VEL
LIN {X 0,Y 452.632,Z 627.243,A -85,B 0,C 180,E1 -8372.671,E2 -8372.671} C_VEL
LIN {X 0,Y 452.609,Z 624.756,A -85,B 0,C 180,E1 -8374.008,E2 -8374.008} C_VEL
LIN {X 0,Y 452.625,Z 621.22,A -85,B 0,C 180,E1 -8375.347,E2 -8375.347} C_VEL
LIN {X 0,Y 452.712,Z 615.991,A -85,B 0,C 180,E1 -8376.833,E2 -8376.833} C_VEL
LIN {X 0,Y 452.832,Z 609.489,A -85,B 0,C 180,E1 -8378.255,E2 -8378.255} C_VEL
LIN {X 0,Y 453.063,Z 601.778,A -85,B 0,C 180,E1 -8379.6,E2 -8379.6} C_VEL
LIN {X 0,Y 453.454,Z 592.215,A -85,B 0,C 180,E1 -8380.946,E2 -8380.946} C_VEL
LIN {X 0,Y 453.796,Z 583.408,A -85,B 0,C 180,E1 -8381.956,E2 -8381.956} C_VEL
LIN {X 0,Y 454.268,Z 572.575,A -85,B 0,C 180,E1 -8382.973,E2 -8382.973} C_VEL
LIN {X 0,Y 454.876,Z 560.823,A -85,B 0,C 180,E1 -8383.857,E2 -8383.857} C_VEL
LIN {X 0,Y 455.414,Z 548.344,A -85,B 0,C 180,E1 -8384.581,E2 -8384.581} C_VEL
LIN {X 0,Y 455.941,Z 534.763,A -85,B 0,C 180,E1 -8385.164,E2 -8385.164} C_VEL
LIN {X 0,Y 456.45,Z 521.03,A -85,B 0,C 180,E1 -8385.547,E2 -8385.547} C_VEL
LIN {X 0,Y 457.527,Z 438.056,A -85,B 0,C 180,E1 -8387.12,E2 -8387.12} C_VEL
LIN {X 0,Y 454.672,Z 415.482,A -85,B 0,C 180,E1 -8387.719,E2 -8387.719} C_VEL
LIN {X 0,Y 454.293,Z 412.967,A -85,B 0,C 180,E1 -8387.793,E2 -8387.793} C_VEL
LIN {X 0,Y 455.11,Z 394.419,A -85,B 0,C 180,E1 -8390.805,E2 -8390.805} C_VEL
LIN {X 0,Y 456.116,Z 376.11,A -85,B 0,C 180,E1 -8393.859,E2 -8393.859} C_VEL
LIN {X 0,Y 456.753,Z 366.407,A -85,B 0,C 180,E1 -8395.521,E2 -8395.521} C_VEL
LIN {X 0,Y 455.751,Z 359.617,A -85,B 0,C 180,E1 -8396.812,E2 -8396.812} C_VEL
LIN {X 0,Y 453.507,Z 349.999,A -85,B 0,C 180,E1 -8398.808,E2 -8398.808} C_VEL
LIN {X 0,Y 453.47,Z 350.001,A -85,B 0,C 180,E1 -8401.8,E2 -8401.8} C_VEL
LIN {X 0,Y 453.486,Z 350.001,A -85,B 0,C 180,E1 -8404.99,E2 -8404.99} C_VEL
LIN {X 0,Y 453.47,Z 349.999,A -85,B 0,C 180,E1 -8408.312,E2 -8408.312} C_VEL
LIN {X 0,Y 453.499,Z 349.997,A -85,B 0,C 180,E1 -8410.609,E2 -8410.609} C_VEL
LIN {X 0,Y 453.461,Z 350.001,A -85,B 0,C 180,E1 -8413.245,E2 -8413.245} C_VEL
LIN {X 0,Y 453.472,Z 349.997,A -85,B 0,C 180,E1 -8415.779,E2 -8415.779} C_VEL
LIN {X 0,Y 453.485,Z 349.994,A -85,B 0,C 180,E1 -8418.21,E2 -8418.21} C_VEL
LIN {X 0,Y 453.515,Z 349.995,A -85,B 0,C 180,E1 -8420.791,E2 -8420.791} C_VEL
LIN {X 0,Y 453.459,Z 349.997,A -85,B 0,C 180,E1 -8423.917,E2 -8423.917} C_VEL
LIN {X 0,Y 453.488,Z 349.998,A -85,B 0,C 180,E1 -8427.151,E2 -8427.151} C_VEL
LIN {X 0,Y 453.48,Z 349.998,A -85,B 0,C 180,E1 -8430.269,E2 -8430.269} C_VEL
LIN {X 0,Y 453.512,Z 349.996,A -85,B 0,C 180,E1 -8433.294,E2 -8433.294} C_VEL
LIN {X 0,Y 453.508,Z 349.995,A -85,B 0,C 180,E1 -8436.239,E2 -8436.239} C_VEL
LIN {X 0,Y 453.488,Z 350,A -85,B 0,C 180,E1 -8439.118,E2 -8439.118} C_VEL
LIN {X 0,Y 453.563,Z 350.058,A -85,B 0,C 180,E1 -8440.734,E2 -8440.734} C_VEL
LIN {X 0,Y 454.656,Z 355.506,A -85,B 0,C 180,E1 -8442.329,E2 -8442.329} C_VEL
LIN {X 0,Y 458.208,Z 365.762,A -85,B 0,C 180,E1 -8442.732,E2 -8442.732} C_VEL
LIN {X 0,Y 457.192,Z 428.242,A -85,B 0,C 180,E1 -8443.965,E2 -8443.965} C_VEL
LIN {X 0,Y 456.728,Z 461.159,A -85,B 0,C 180,E1 -8444.607,E2 -8444.607} C_VEL
LIN {X 0,Y 456.457,Z 474.721,A -85,B 0,C 180,E1 -8445.055,E2 -8445.055} C_VEL
LIN {X 0,Y 456.087,Z 486.525,A -85,B 0,C 180,E1 -8445.613,E2 -8445.613} C_VEL
LIN {X 0,Y 455.717,Z 498.683,A -85,B 0,C 180,E1 -8446.385,E2 -8446.385} C_VEL
LIN {X 0,Y 455.186,Z 509.91,A -85,B 0,C 180,E1 -8447.29,E2 -8447.29} C_VEL
LIN {X 0,Y 454.764,Z 518.863,A -85,B 0,C 180,E1 -8448.184,E2 -8448.184} C_VEL
LIN {X 0,Y 454.357,Z 528.034,A -85,B 0,C 180,E1 -8449.303,E2 -8449.303} C_VEL
LIN {X 0,Y 453.869,Z 536.936,A -85,B 0,C 180,E1 -8450.643,E2 -8450.643} C_VEL
LIN {X 0,Y 453.51,Z 544.061,A -85,B 0,C 180,E1 -8451.983,E2 -8451.983} C_VEL
LIN {X 0,Y 453.158,Z 549.695,A -85,B 0,C 180,E1 -8453.319,E2 -8453.319} C_VEL
LIN {X 0,Y 453.093,Z 554.086,A -85,B 0,C 180,E1 -8454.66,E2 -8454.66} C_VEL
LIN {X 0,Y 452.935,Z 556.399,A -85,B 0,C 180,E1 -8455.55,E2 -8455.55} C_VEL
LIN {X 0,Y 452.919,Z 558.264,A -85,B 0,C 180,E1 -8456.441,E2 -8456.441} C_VEL
LIN {X 0,Y 452.745,Z 559.679,A -85,B 0,C 180,E1 -8457.331,E2 -8457.331} C_VEL
LIN {X 0,Y 452.6,Z 560.655,A -85,B 0,C 180,E1 -8458.22,E2 -8458.22} C_VEL
LIN {X 0,Y 452.531,Z 561.227,A -85,B 0,C 180,E1 -8459.11,E2 -8459.11} C_VEL
LIN {X 0,Y 452.514,Z 561.394,A -85,B 0,C 180,E1 -8460,E2 -8460} C_VEL
LIN {X 0,Y 452.528,Z 561.107,A -85,B 0,C 180,E1 -8460.89,E2 -8460.89} C_VEL
LIN {X 0,Y 452.595,Z 560.414,A -85,B 0,C 180,E1 -8461.78,E2 -8461.78} C_VEL
LIN {X 0,Y 452.738,Z 559.32,A -85,B 0,C 180,E1 -8462.669,E2 -8462.669} C_VEL
LIN {X 0,Y 452.828,Z 557.797,A -85,B 0,C 180,E1 -8463.559,E2 -8463.559} C_VEL
LIN {X 0,Y 452.912,Z 554.677,A -85,B 0,C 180,E1 -8464.896,E2 -8464.896} C_VEL
LIN {X 0,Y 453.025,Z 550.472,A -85,B 0,C 180,E1 -8466.234,E2 -8466.234} C_VEL
LIN {X 0,Y 453.256,Z 544.021,A -85,B 0,C 180,E1 -8467.798,E2 -8467.798} C_VEL
LIN {X 0,Y 453.606,Z 536.991,A -85,B 0,C 180,E1 -8469.138,E2 -8469.138} C_VEL
LIN {X 0,Y 453.996,Z 528.167,A -85,B 0,C 180,E1 -8470.48,E2 -8470.48} C_VEL
LIN {X 0,Y 454.469,Z 518.114,A -85,B 0,C 180,E1 -8471.71,E2 -8471.71} C_VEL
LIN {X 0,Y 454.983,Z 508.072,A -85,B 0,C 180,E1 -8472.7,E2 -8472.7} C_VEL
LIN {X 0,Y 455.293,Z 497.133,A -85,B 0,C 180,E1 -8473.572,E2 -8473.572} C_VEL
LIN {X 0,Y 455.724,Z 484.818,A -85,B 0,C 180,E1 -8474.342,E2 -8474.342} C_VEL
LIN {X 0,Y 456.154,Z 472.168,A -85,B 0,C 180,E1 -8474.927,E2 -8474.927} C_VEL
LIN {X 0,Y 456.422,Z 460.12,A -85,B 0,C 180,E1 -8475.318,E2 -8475.318} C_VEL
LIN {X 0,Y 456.622,Z 436.807,A -85,B 0,C 180,E1 -8475.769,E2 -8475.769} C_VEL
LIN {X 0,Y 457.41,Z 364.774,A -85,B 0,C 180,E1 -8477.068,E2 -8477.068} C_VEL
LIN {X 0,Y 454.618,Z 354.144,A -85,B 0,C 180,E1 -8477.368,E2 -8477.368} C_VEL
LIN {X 0,Y 453.743,Z 351.101,A -85,B 0,C 180,E1 -8477.468,E2 -8477.468} C_VEL
LIN {X 0,Y 453.548,Z 349.991,A -85,B 0,C 180,E1 -8477.763,E2 -8477.763} C_VEL
LIN {X 0,Y 453.487,Z 349.998,A -85,B 0,C 180,E1 -8480.882,E2 -8480.882} C_VEL
LIN {X 0,Y 453.502,Z 349.995,A -85,B 0,C 180,E1 -8483.887,E2 -8483.887} C_VEL
LIN {X 0,Y 453.509,Z 349.994,A -85,B 0,C 180,E1 -8486.706,E2 -8486.706} C_VEL
LIN {X 0,Y 453.477,Z 349.998,A -85,B 0,C 180,E1 -8489.784,E2 -8489.784} C_VEL
LIN {X 0,Y 453.495,Z 349.996,A -85,B 0,C 180,E1 -8493.189,E2 -8493.189} C_VEL
LIN {X 0,Y 453.457,Z 349.999,A -85,B 0,C 180,E1 -8496.299,E2 -8496.299} C_VEL
LIN {X 0,Y 453.51,Z 349.994,A -85,B 0,C 180,E1 -8499.448,E2 -8499.448} C_VEL
LIN {X 0,Y 453.468,Z 350,A -85,B 0,C 180,E1 -8502.994,E2 -8502.994} C_VEL
LIN {X 0,Y 453.47,Z 349.998,A -85,B 0,C 180,E1 -8505.779,E2 -8505.779} C_VEL
LIN {X 0,Y 453.483,Z 349.996,A -85,B 0,C 180,E1 -8508.209,E2 -8508.209} C_VEL
LIN {X 0,Y 453.514,Z 349.995,A -85,B 0,C 180,E1 -8510.79,E2 -8510.79} C_VEL
LIN {X 0,Y 453.459,Z 349.999,A -85,B 0,C 180,E1 -8513.917,E2 -8513.917} C_VEL
LIN {X 0,Y 453.487,Z 349.997,A -85,B 0,C 180,E1 -8517.151,E2 -8517.151} C_VEL
LIN {X 0,Y 453.479,Z 349.997,A -85,B 0,C 180,E1 -8520.268,E2 -8520.268} C_VEL
LIN {X 0,Y 453.511,Z 349.994,A -85,B 0,C 180,E1 -8523.293,E2 -8523.293} C_VEL
LIN {X 0,Y 453.508,Z 349.994,A -85,B 0,C 180,E1 -8526.238,E2 -8526.238} C_VEL
LIN {X 0,Y 453.47,Z 349.997,A -85,B 0,C 180,E1 -8527.958,E2 -8527.958} C_VEL
LIN {X 0,Y 452.831,Z 350.08,A -85,B 0,C 180,E1 -8528.699,E2 -8528.699} C_VEL
LIN {X 0,Y 449.998,Z 350.433,A -85,B 0,C 180,E1 -8529.904,E2 -8529.904} C_VEL
LIN {X 0,Y 447.582,Z 350.732,A -85,B 0,C 180,E1 -8530.875,E2 -8530.875} C_VEL
LIN {X 0,Y 446.539,Z 350.861,A -85,B 0,C 180,E1 -8531.626,E2 -8531.626} C_VEL
LIN {X 0,Y 446.451,Z 350.871,A -85,B 0,C 180,E1 -8531.88,E2 -8531.88} C_VEL
LIN {X 0,Y 446.511,Z 350.868,A -85,B 0,C 180,E1 -8534.479,E2 -8534.479} C_VEL
LIN {X 0,Y 446.521,Z 350.865,A -85,B 0,C 180,E1 -8538.192,E2 -8538.192} C_VEL
LIN {X 0,Y 446.603,Z 350.853,A -85,B 0,C 180,E1 -8541.857,E2 -8541.857} C_VEL
LIN {X 0,Y 446.645,Z 350.85,A -85,B 0,C 180,E1 -8544.582,E2 -8544.582} C_VEL
LIN {X 0,Y 446.712,Z 350.839,A -85,B 0,C 180,E1 -8547.294,E2 -8547.294} C_VEL
LIN {X 0,Y 446.796,Z 350.83,A -85,B 0,C 180,E1 -8549.999,E2 -8549.999} C_VEL
LIN {X 0,Y 446.711,Z 350.84,A -85,B 0,C 180,E1 -8552.704,E2 -8552.704} C_VEL
LIN {X 0,Y 446.649,Z 350.851,A -85,B 0,C 180,E1 -8556.323,E2 -8556.323} C_VEL
LIN {X 0,Y 446.539,Z 350.861,A -85,B 0,C 180,E1 -8559.054,E2 -8559.054} C_VEL
LIN {X 0,Y 446.521,Z 350.864,A -85,B 0,C 180,E1 -8562.729,E2 -8562.729} C_VEL
LIN {X 0,Y 446.518,Z 350.867,A -85,B 0,C 180,E1 -8566.237,E2 -8566.237} C_VEL
LIN {X 0,Y 446.468,Z 350.869,A -85,B 0,C 180,E1 -8569.302,E2 -8569.302} C_VEL
LIN {X 0,Y 446.417,Z 350.88,A -85,B 0,C 180,E1 -8572.198,E2 -8572.198} C_VEL
LIN {X 0,Y 446.456,Z 350.87,A -85,B 0,C 180,E1 -8575.151,E2 -8575.151} C_VEL
LIN {X 0,Y 446.481,Z 350.871,A -85,B 0,C 180,E1 -8578.177,E2 -8578.177} C_VEL
LIN {X 0,Y 446.416,Z 350.875,A -85,B 0,C 180,E1 -8581.299,E2 -8581.299} C_VEL
LIN {X 0,Y 446.426,Z 350.875,A -85,B 0,C 180,E1 -8584.522,E2 -8584.522} C_VEL
LIN {X 0,Y 446.434,Z 350.877,A -85,B 0,C 180,E1 -8588.082,E2 -8588.082} C_VEL
LIN {X 0,Y 446.442,Z 350.872,A -85,B 0,C 180,E1 -8590.92,E2 -8590.92} C_VEL
LIN {X 0,Y 446.439,Z 350.877,A -85,B 0,C 180,E1 -8593.839,E2 -8593.839} C_VEL
LIN {X 0,Y 446.44,Z 350.873,A -85,B 0,C 180,E1 -8596.396,E2 -8596.396} C_VEL
LIN {X 0,Y 446.463,Z 350.874,A -85,B 0,C 180,E1 -8599.804,E2 -8599.804} C_VEL
LIN {X 0,Y 446.427,Z 350.876,A -85,B 0,C 180,E1 -8602.123,E2 -8602.123} C_VEL
LIN {X 0,Y 446.423,Z 350.876,A -85,B 0,C 180,E1 -8605.476,E2 -8605.476} C_VEL
LIN {X 0,Y 446.411,Z 350.875,A -85,B 0,C 180,E1 -8608.699,E2 -8608.699} C_VEL
LIN {X 0,Y 446.475,Z 350.873,A -85,B 0,C 180,E1 -8611.821,E2 -8611.821} C_VEL
LIN {X 0,Y 446.449,Z 350.87,A -85,B 0,C 180,E1 -8614.847,E2 -8614.847} C_VEL
LIN {X 0,Y 446.439,Z 350.873,A -85,B 0,C 180,E1 -8618.244,E2 -8618.244} C_VEL
LIN {X 0,Y 446.449,Z 350.877,A -85,B 0,C 180,E1 -8621.649,E2 -8621.649} C_VEL
LIN {X 0,Y 446.506,Z 350.863,A -85,B 0,C 180,E1 -8624.48,E2 -8624.48} C_VEL
LIN {X 0,Y 446.53,Z 350.861,A -85,B 0,C 180,E1 -8628.193,E2 -8628.193} C_VEL
LIN {X 0,Y 446.59,Z 350.856,A -85,B 0,C 180,E1 -8631.858,E2 -8631.858} C_VEL
LIN {X 0,Y 446.637,Z 350.846,A -85,B 0,C 180,E1 -8634.583,E2 -8634.583} C_VEL
LIN {X 0,Y 446.701,Z 350.842,A -85,B 0,C 180,E1 -8637.295,E2 -8637.295} C_VEL
LIN {X 0,Y 446.785,Z 350.829,A -85,B 0,C 180,E1 -8640,E2 -8640} C_VEL
LIN {X 0,Y 446.701,Z 350.838,A -85,B 0,C 180,E1 -8642.705,E2 -8642.705} C_VEL
LIN {X 0,Y 446.642,Z 350.845,A -85,B 0,C 180,E1 -8646.324,E2 -8646.324} C_VEL
LIN {X 0,Y 446.53,Z 350.862,A -85,B 0,C 180,E1 -8649.056,E2 -8649.056} C_VEL
LIN {X 0,Y 446.525,Z 350.861,A -85,B 0,C 180,E1 -8652.73,E2 -8652.73} C_VEL
LIN {X 0,Y 446.481,Z 350.865,A -85,B 0,C 180,E1 -8656.46,E2 -8656.46} C_VEL
LIN {X 0,Y 446.46,Z 350.875,A -85,B 0,C 180,E1 -8659.304,E2 -8659.304} C_VEL
LIN {X 0,Y 446.409,Z 350.874,A -85,B 0,C 180,E1 -8662.2,E2 -8662.2} C_VEL
LIN {X 0,Y 446.45,Z 350.875,A -85,B 0,C 180,E1 -8665.153,E2 -8665.153} C_VEL
LIN {X 0,Y 446.476,Z 350.866,A -85,B 0,C 180,E1 -8668.179,E2 -8668.179} C_VEL
LIN {X 0,Y 446.412,Z 350.876,A -85,B 0,C 180,E1 -8671.776,E2 -8671.776} C_VEL
LIN {X 0,Y 446.423,Z 350.874,A -85,B 0,C 180,E1 -8674.524,E2 -8674.524} C_VEL
LIN {X 0,Y 446.432,Z 350.872,A -85,B 0,C 180,E1 -8678.084,E2 -8678.084} C_VEL
LIN {X 0,Y 446.442,Z 350.875,A -85,B 0,C 180,E1 -8680.922,E2 -8680.922} C_VEL
LIN {X 0,Y 446.44,Z 350.872,A -85,B 0,C 180,E1 -8683.841,E2 -8683.841} C_VEL
LIN {X 0,Y 446.442,Z 350.872,A -85,B 0,C 180,E1 -8686.398,E2 -8686.398} C_VEL
LIN {X 0,Y 446.464,Z 350.869,A -85,B 0,C 180,E1 -8689.806,E2 -8689.806} C_VEL
LIN {X 0,Y 446.431,Z 350.873,A -85,B 0,C 180,E1 -8692.125,E2 -8692.125} C_VEL
LIN {X 0,Y 446.427,Z 350.875,A -85,B 0,C 180,E1 -8695.478,E2 -8695.478} C_VEL
LIN {X 0,Y 446.431,Z 350.878,A -85,B 0,C 180,E1 -8698.702,E2 -8698.702} C_VEL
LIN {X 0,Y 446.502,Z 350.959,A -85,B 0,C 180,E1 -8701.335,E2 -8701.335} C_VEL
LIN {X 0,Y 449.628,Z 365.857,A -85,B 0,C 180,E1 -8704.047,E2 -8704.047} C_VEL
LIN {X 0,Y 449.568,Z 372.533,A -85,B 0,C 180,E1 -8705.17,E2 -8705.17} C_VEL
LIN {X 0,Y 448.492,Z 392.118,A -85,B 0,C 180,E1 -8708.393,E2 -8708.393} C_VEL
LIN {X 0,Y 447.486,Z 414.019,A -85,B 0,C 180,E1 -8711.955,E2 -8711.955} C_VEL
LIN {X 0,Y 447.431,Z 416.231,A -85,B 0,C 180,E1 -8712.279,E2 -8712.279} C_VEL
LIN {X 0,Y 450.381,Z 439.656,A -85,B 0,C 180,E1 -8712.831,E2 -8712.831} C_VEL
LIN {X 0,Y 449.268,Z 525.837,A -85,B 0,C 180,E1 -8714.433,E2 -8714.433} C_VEL
LIN {X 0,Y 448.778,Z 539.807,A -85,B 0,C 180,E1 -8714.881,E2 -8714.881} C_VEL
LIN {X 0,Y 448.291,Z 552.355,A -85,B 0,C 180,E1 -8715.474,E2 -8715.474} C_VEL
LIN {X 0,Y 447.735,Z 564.827,A -85,B 0,C 180,E1 -8716.267,E2 -8716.267} C_VEL
LIN {X 0,Y 447.202,Z 575.884,A -85,B 0,C 180,E1 -8717.162,E2 -8717.162} C_VEL
LIN {X 0,Y 446.7,Z 586.147,A -85,B 0,C 180,E1 -8718.199,E2 -8718.199} C_VEL
LIN {X 0,Y 446.295,Z 595.333,A -85,B 0,C 180,E1 -8719.338,E2 -8719.338} C_VEL
LIN {X 0,Y 445.932,Z 604.298,A -85,B 0,C 180,E1 -8720.705,E2 -8720.705} C_VEL
LIN {X 0,Y 445.701,Z 611.428,A -85,B 0,C 180,E1 -8722.071,E2 -8722.071} C_VEL
LIN {X 0,Y 445.578,Z 617.947,A -85,B 0,C 180,E1 -8723.662,E2 -8723.662} C_VEL
LIN {X 0,Y 445.507,Z 622.188,A -85,B 0,C 180,E1 -8725.024,E2 -8725.024} C_VEL
LIN {X 0,Y 445.543,Z 625.316,A -85,B 0,C 180,E1 -8726.384,E2 -8726.384} C_VEL
LIN {X 0,Y 445.533,Z 626.836,A -85,B 0,C 180,E1 -8727.289,E2 -8727.289} C_VEL
LIN {X 0,Y 445.518,Z 627.877,A -85,B 0,C 180,E1 -8728.193,E2 -8728.193} C_VEL
LIN {X 0,Y 445.441,Z 628.497,A -85,B 0,C 180,E1 -8729.097,E2 -8729.097} C_VEL
LIN {X 0,Y 445.427,Z 628.71,A -85,B 0,C 180,E1 -8730.001,E2 -8730.001} C_VEL
LIN {X 0,Y 445.443,Z 628.475,A -85,B 0,C 180,E1 -8730.905,E2 -8730.905} C_VEL
LIN {X 0,Y 445.521,Z 627.802,A -85,B 0,C 180,E1 -8731.809,E2 -8731.809} C_VEL
LIN {X 0,Y 445.553,Z 626.711,A -85,B 0,C 180,E1 -8732.713,E2 -8732.713} C_VEL
LIN {X 0,Y 445.505,Z 624.224,A -85,B 0,C 180,E1 -8734.072,E2 -8734.072} C_VEL
LIN {X 0,Y 445.538,Z 620.688,A -85,B 0,C 180,E1 -8735.432,E2 -8735.432} C_VEL
LIN {X 0,Y 445.634,Z 615.228,A -85,B 0,C 180,E1 -8736.999,E2 -8736.999} C_VEL
LIN {X 0,Y 445.766,Z 608.948,A -85,B 0,C 180,E1 -8738.387,E2 -8738.387} C_VEL
LIN {X 0,Y 445.982,Z 601.237,A -85,B 0,C 180,E1 -8739.754,E2 -8739.754} C_VEL
LIN {X 0,Y 446.421,Z 591.683,A -85,B 0,C 180,E1 -8741.12,E2 -8741.12} C_VEL
LIN {X 0,Y 446.835,Z 582.88,A -85,B 0,C 180,E1 -8742.145,E2 -8742.145} C_VEL
LIN {X 0,Y 447.334,Z 571.604,A -85,B 0,C 180,E1 -8743.219,E2 -8743.219} C_VEL
LIN {X 0,Y 447.955,Z 560.365,A -85,B 0,C 180,E1 -8744.075,E2 -8744.075} C_VEL
LIN {X 0,Y 448.536,Z 547.997,A -85,B 0,C 180,E1 -8744.81,E2 -8744.81} C_VEL
LIN {X 0,Y 449.12,Z 533.813,A -85,B 0,C 180,E1 -8745.429,E2 -8745.429} C_VEL
LIN {X 0,Y 449.651,Z 519.998,A -85,B 0,C 180,E1 -8745.817,E2 -8745.817} C_VEL
LIN {X 0,Y 450.859,Z 438.951,A -85,B 0,C 180,E1 -8747.402,E2 -8747.402} C_VEL
LIN {X 0,Y 448.073,Z 416.689,A -85,B 0,C 180,E1 -8748.018,E2 -8748.018} C_VEL
LIN {X 0,Y 447.365,Z 412.148,A -85,B 0,C 180,E1 -8748.165,E2 -8748.165} C_VEL
LIN {X 0,Y 448.351,Z 392.816,A -85,B 0,C 180,E1 -8751.375,E2 -8751.375} C_VEL
LIN {X 0,Y 449.439,Z 374.726,A -85,B 0,C 180,E1 -8754.478,E2 -8754.478} C_VEL
LIN {X 0,Y 449.923,Z 367.873,A -85,B 0,C 180,E1 -8755.688,E2 -8755.688} C_VEL
LIN {X 0,Y 448.601,Z 359.816,A -85,B 0,C 180,E1 -8757.275,E2 -8757.275} C_VEL
LIN {X 0,Y 446.496,Z 350.872,A -85,B 0,C 180,E1 -8759.207,E2 -8759.207} C_VEL
LIN {X 0,Y 446.428,Z 350.878,A -85,B 0,C 180,E1 -8762.362,E2 -8762.362} C_VEL
LIN {X 0,Y 446.425,Z 350.878,A -85,B 0,C 180,E1 -8765.626,E2 -8765.626} C_VEL
LIN {X 0,Y 446.461,Z 350.875,A -85,B 0,C 180,E1 -8769.026,E2 -8769.026} C_VEL
LIN {X 0,Y 446.44,Z 350.873,A -85,B 0,C 180,E1 -8772.278,E2 -8772.278} C_VEL
LIN {X 0,Y 446.459,Z 350.873,A -85,B 0,C 180,E1 -8775.104,E2 -8775.104} C_VEL
LIN {X 0,Y 446.434,Z 350.875,A -85,B 0,C 180,E1 -8778.609,E2 -8778.609} C_VEL
LIN {X 0,Y 446.461,Z 350.873,A -85,B 0,C 180,E1 -8780.974,E2 -8780.974} C_VEL
LIN {X 0,Y 446.424,Z 350.875,A -85,B 0,C 180,E1 -8784.374,E2 -8784.374} C_VEL
LIN {X 0,Y 446.428,Z 350.875,A -85,B 0,C 180,E1 -8787.639,E2 -8787.639} C_VEL
LIN {X 0,Y 446.454,Z 350.875,A -85,B 0,C 180,E1 -8790.791,E2 -8790.791} C_VEL
LIN {X 0,Y 446.483,Z 350.869,A -85,B 0,C 180,E1 -8793.849,E2 -8793.849} C_VEL
LIN {X 0,Y 446.434,Z 350.878,A -85,B 0,C 180,E1 -8796.823,E2 -8796.823} C_VEL
LIN {X 0,Y 446.489,Z 350.871,A -85,B 0,C 180,E1 -8800.279,E2 -8800.279} C_VEL
LIN {X 0,Y 447.653,Z 356.43,A -85,B 0,C 180,E1 -8801.97,E2 -8801.97} C_VEL
LIN {X 0,Y 451.681,Z 367.316,A -85,B 0,C 180,E1 -8802.432,E2 -8802.432} C_VEL
LIN {X 0,Y 450.165,Z 451.14,A -85,B 0,C 180,E1 -8804.115,E2 -8804.115} C_VEL
LIN {X 0,Y 449.908,Z 465.715,A -85,B 0,C 180,E1 -8804.455,E2 -8804.455} C_VEL
LIN {X 0,Y 449.588,Z 478.461,A -85,B 0,C 180,E1 -8804.937,E2 -8804.937} C_VEL
LIN {X 0,Y 449.158,Z 491.463,A -85,B 0,C 180,E1 -8805.624,E2 -8805.624} C_VEL
LIN {X 0,Y 448.735,Z 502.716,A -85,B 0,C 180,E1 -8806.413,E2 -8806.413} C_VEL
LIN {X 0,Y 448.137,Z 514.218,A -85,B 0,C 180,E1 -8807.432,E2 -8807.432} C_VEL
LIN {X 0,Y 447.622,Z 523.522,A -85,B 0,C 180,E1 -8808.452,E2 -8808.452} C_VEL
LIN {X 0,Y 447.24,Z 531.963,A -85,B 0,C 180,E1 -8809.589,E2 -8809.589} C_VEL
LIN {X 0,Y 446.788,Z 540.162,A -85,B 0,C 180,E1 -8810.95,E2 -8810.95} C_VEL
LIN {X 0,Y 446.378,Z 546.74,A -85,B 0,C 180,E1 -8812.309,E2 -8812.309} C_VEL
LIN {X 0,Y 446.004,Z 551.96,A -85,B 0,C 180,E1 -8813.667,E2 -8813.667} C_VEL
LIN {X 0,Y 445.965,Z 555.957,A -85,B 0,C 180,E1 -8815.028,E2 -8815.028} C_VEL
LIN {X 0,Y 445.877,Z 558.88,A -85,B 0,C 180,E1 -8816.385,E2 -8816.385} C_VEL
LIN {X 0,Y 445.697,Z 560.274,A -85,B 0,C 180,E1 -8817.288,E2 -8817.288} C_VEL
LIN {X 0,Y 445.543,Z 561.237,A -85,B 0,C 180,E1 -8818.192,E2 -8818.192} C_VEL
LIN {X 0,Y 445.467,Z 561.796,A -85,B 0,C 180,E1 -8819.096,E2 -8819.096} C_VEL
LIN {X 0,Y 445.447,Z 561.941,A -85,B 0,C 180,E1 -8820,E2 -8820} C_VEL
LIN {X 0,Y 445.464,Z 561.632,A -85,B 0,C 180,E1 -8820.904,E2 -8820.904} C_VEL
LIN {X 0,Y 445.539,Z 560.92,A -85,B 0,C 180,E1 -8821.808,E2 -8821.808} C_VEL
LIN {X 0,Y 445.688,Z 559.805,A -85,B 0,C 180,E1 -8822.711,E2 -8822.711} C_VEL
LIN {X 0,Y 445.786,Z 557.308,A -85,B 0,C 180,E1 -8824.068,E2 -8824.068} C_VEL
LIN {X 0,Y 445.788,Z 553.796,A -85,B 0,C 180,E1 -8825.428,E2 -8825.428} C_VEL
LIN {X 0,Y 446.1,Z 548.274,A -85,B 0,C 180,E1 -8827.007,E2 -8827.007} C_VEL
LIN {X 0,Y 446.383,Z 540.955,A -85,B 0,C 180,E1 -8828.602,E2 -8828.602} C_VEL
LIN {X 0,Y 446.788,Z 532.994,A -85,B 0,C 180,E1 -8829.964,E2 -8829.964} C_VEL
LIN {X 0,Y 447.276,Z 523.022,A -85,B 0,C 180,E1 -8831.327,E2 -8831.327} C_VEL
LIN {X 0,Y 447.774,Z 512.629,A -85,B 0,C 180,E1 -8832.463,E2 -8832.463} C_VEL
LIN {X 0,Y 448.237,Z 501.311,A -85,B 0,C 180,E1 -8833.453,E2 -8833.453} C_VEL
LIN {X 0,Y 448.602,Z 491.105,A -85,B 0,C 180,E1 -8834.169,E2 -8834.169} C_VEL
LIN {X 0,Y 449.014,Z 478.636,A -85,B 0,C 180,E1 -8834.851,E2 -8834.851} C_VEL
LIN {X 0,Y 449.331,Z 465.541,A -85,B 0,C 180,E1 -8835.362,E2 -8835.362} C_VEL
LIN {X 0,Y 449.615,Z 451.931,A -85,B 0,C 180,E1 -8835.701,E2 -8835.701} C_VEL
LIN {X 0,Y 450.607,Z 366.013,A -85,B 0,C 180,E1 -8837.281,E2 -8837.281} C_VEL
LIN {X 0,Y 447.739,Z 355.293,A -85,B 0,C 180,E1 -8837.592,E2 -8837.592} C_VEL
LIN {X 0,Y 446.616,Z 351.476,A -85,B 0,C 180,E1 -8837.732,E2 -8837.732} C_VEL
LIN {X 0,Y 446.505,Z 350.868,A -85,B 0,C 180,E1 -8837.933,E2 -8837.933} C_VEL
LIN {X 0,Y 446.458,Z 350.873,A -85,B 0,C 180,E1 -8841.227,E2 -8841.227} C_VEL
LIN {X 0,Y 446.47,Z 350.87,A -85,B 0,C 180,E1 -8844.159,E2 -8844.159} C_VEL
LIN {X 0,Y 446.478,Z 350.87,A -85,B 0,C 180,E1 -8847.161,E2 -8847.161} C_VEL
LIN {X 0,Y 446.432,Z 350.874,A -85,B 0,C 180,E1 -8850.249,E2 -8850.249} C_VEL
LIN {X 0,Y 446.45,Z 350.874,A -85,B 0,C 180,E1 -8853.453,E2 -8853.453} C_VEL
LIN {X 0,Y 446.406,Z 350.881,A -85,B 0,C 180,E1 -8856.745,E2 -8856.745} C_VEL
LIN {X 0,Y 446.452,Z 350.872,A -85,B 0,C 180,E1 -8860.197,E2 -8860.197} C_VEL
LIN {X 0,Y 446.434,Z 350.876,A -85,B 0,C 180,E1 -8862.604,E2 -8862.604} C_VEL
LIN {X 0,Y 446.458,Z 350.872,A -85,B 0,C 180,E1 -8865.103,E2 -8865.103} C_VEL
LIN {X 0,Y 446.432,Z 350.877,A -85,B 0,C 180,E1 -8868.608,E2 -8868.608} C_VEL
LIN {X 0,Y 446.46,Z 350.872,A -85,B 0,C 180,E1 -8870.974,E2 -8870.974} C_VEL
LIN {X 0,Y 446.424,Z 350.877,A -85,B 0,C 180,E1 -8874.373,E2 -8874.373} C_VEL
LIN {X 0,Y 446.426,Z 350.875,A -85,B 0,C 180,E1 -8877.638,E2 -8877.638} C_VEL
LIN {X 0,Y 446.453,Z 350.874,A -85,B 0,C 180,E1 -8880.79,E2 -8880.79} C_VEL
LIN {X 0,Y 446.482,Z 350.868,A -85,B 0,C 180,E1 -8883.848,E2 -8883.848} C_VEL
LIN {X 0,Y 446.433,Z 350.876,A -85,B 0,C 180,E1 -8886.823,E2 -8886.823} C_VEL
LIN {X 0,Y 446.448,Z 350.872,A -85,B 0,C 180,E1 -8889.736,E2 -8889.736} C_VEL
LIN {X 0,Y 446.451,Z 350.871,A -85,B 0,C 180,E1 -8891.88,E2 -8891.88} C_VEL
LIN {X 0,Y 445.778,Z 350.958,A -85,B 0,C 180,E1 -8892.633,E2 -8892.633} C_VEL
LIN {X 0,Y 442.928,Z 351.311,A -85,B 0,C 180,E1 -8893.857,E2 -8893.857} C_VEL
LIN {X 0,Y 440.526,Z 351.611,A -85,B 0,C 180,E1 -8894.845,E2 -8894.845} C_VEL
LIN {X 0,Y 439.501,Z 351.737,A -85,B 0,C 180,E1 -8895.607,E2 -8895.607} C_VEL
LIN {X 0,Y 439.421,Z 351.747,A -85,B 0,C 180,E1 -8895.866,E2 -8895.866} C_VEL
LIN {X 0,Y 439.487,Z 351.74,A -85,B 0,C 180,E1 -8898,E2 -8898} C_VEL
LIN {X 0,Y 439.551,Z 351.731,A -85,B 0,C 180,E1 -8901.725,E2 -8901.725} C_VEL
LIN {X 0,Y 439.62,Z 351.726,A -85,B 0,C 180,E1 -8904.495,E2 -8904.495} C_VEL
LIN {X 0,Y 439.639,Z 351.723,A -85,B 0,C 180,E1 -8908.167,E2 -8908.167} C_VEL
LIN {X 0,Y 439.766,Z 351.706,A -85,B 0,C 180,E1 -8909.999,E2 -8909.999} C_VEL
LIN {X 0,Y 439.658,Z 351.719,A -85,B 0,C 180,E1 -8912.748,E2 -8912.748} C_VEL
LIN {X 0,Y 439.62,Z 351.725,A -85,B 0,C 180,E1 -8916.424,E2 -8916.424} C_VEL
LIN {X 0,Y 439.501,Z 351.737,A -85,B 0,C 180,E1 -8919.2,E2 -8919.2} C_VEL
LIN {X 0,Y 439.466,Z 351.742,A -85,B 0,C 180,E1 -8922.936,E2 -8922.936} C_VEL
LIN {X 0,Y 439.46,Z 351.745,A -85,B 0,C 180,E1 -8926.354,E2 -8926.354} C_VEL
LIN {X 0,Y 439.401,Z 351.75,A -85,B 0,C 180,E1 -8929.625,E2 -8929.625} C_VEL
LIN {X 0,Y 439.363,Z 351.755,A -85,B 0,C 180,E1 -8932.574,E2 -8932.574} C_VEL
LIN {X 0,Y 439.403,Z 351.75,A -85,B 0,C 180,E1 -8935.584,E2 -8935.584} C_VEL
LIN {X 0,Y 439.422,Z 351.747,A -85,B 0,C 180,E1 -8938.672,E2 -8938.672} C_VEL
LIN {X 0,Y 439.379,Z 351.757,A -85,B 0,C 180,E1 -8942.032,E2 -8942.032} C_VEL
LIN {X 0,Y 439.392,Z 351.75,A -85,B 0,C 180,E1 -8945.34,E2 -8945.34} C_VEL
LIN {X 0,Y 439.395,Z 351.75,A -85,B 0,C 180,E1 -8948.592,E2 -8948.592} C_VEL
LIN {X 0,Y 439.399,Z 351.749,A -85,B 0,C 180,E1 -8951.258,E2 -8951.258} C_VEL
LIN {X 0,Y 439.403,Z 351.749,A -85,B 0,C 180,E1 -8954.727,E2 -8954.727} C_VEL
LIN {X 0,Y 439.406,Z 351.753,A -85,B 0,C 180,E1 -8957.797,E2 -8957.797} C_VEL
LIN {X 0,Y 439.447,Z 351.745,A -85,B 0,C 180,E1 -8960.23,E2 -8960.23} C_VEL
LIN {X 0,Y 439.369,Z 351.757,A -85,B 0,C 180,E1 -8963.712,E2 -8963.712} C_VEL
LIN {X 0,Y 439.364,Z 351.753,A -85,B 0,C 180,E1 -8967.053,E2 -8967.053} C_VEL
LIN {X 0,Y 439.388,Z 351.751,A -85,B 0,C 180,E1 -8970.275,E2 -8970.275} C_VEL
LIN {X 0,Y 439.424,Z 351.75,A -85,B 0,C 180,E1 -8973.588,E2 -8973.588} C_VEL
LIN {X 0,Y 439.378,Z 351.751,A -85,B 0,C 180,E1 -8976.429,E2 -8976.429} C_VEL
LIN {X 0,Y 439.379,Z 351.754,A -85,B 0,C 180,E1 -8979.397,E2 -8979.397} C_VEL
LIN {X 0,Y 439.423,Z 351.746,A -85,B 0,C 180,E1 -8982.309,E2 -8982.309} C_VEL
LIN {X 0,Y 439.442,Z 351.744,A -85,B 0,C 180,E1 -8985.174,E2 -8985.174} C_VEL
LIN {X 0,Y 439.498,Z 351.738,A -85,B 0,C 180,E1 -8988.002,E2 -8988.002} C_VEL
LIN {X 0,Y 439.538,Z 351.736,A -85,B 0,C 180,E1 -8991.726,E2 -8991.726} C_VEL
LIN {X 0,Y 439.612,Z 351.721,A -85,B 0,C 180,E1 -8994.496,E2 -8994.496} C_VEL
LIN {X 0,Y 439.626,Z 351.72,A -85,B 0,C 180,E1 -8998.168,E2 -8998.168} C_VEL
LIN {X 0,Y 439.755,Z 351.705,A -85,B 0,C 180,E1 -9000,E2 -9000} C_VEL
LIN {X 0,Y 439.648,Z 351.717,A -85,B 0,C 180,E1 -9002.749,E2 -9002.749} C_VEL
LIN {X 0,Y 439.612,Z 351.721,A -85,B 0,C 180,E1 -9006.425,E2 -9006.425} C_VEL
LIN {X 0,Y 439.492,Z 351.74,A -85,B 0,C 180,E1 -9009.202,E2 -9009.202} C_VEL
LIN {X 0,Y 439.495,Z 351.736,A -85,B 0,C 180,E1 -9012.727,E2 -9012.727} C_VEL
LIN {X 0,Y 439.438,Z 351.743,A -85,B 0,C 180,E1 -9016.349,E2 -9016.349} C_VEL
LIN {X 0,Y 439.393,Z 351.752,A -85,B 0,C 180,E1 -9019.627,E2 -9019.627} C_VEL
LIN {X 0,Y 439.357,Z 351.754,A -85,B 0,C 180,E1 -9022.576,E2 -9022.576} C_VEL
LIN {X 0,Y 439.397,Z 351.752,A -85,B 0,C 180,E1 -9025.586,E2 -9025.586} C_VEL
LIN {X 0,Y 439.409,Z 351.748,A -85,B 0,C 180,E1 -9028.674,E2 -9028.674} C_VEL
LIN {X 0,Y 439.363,Z 351.753,A -85,B 0,C 180,E1 -9032.032,E2 -9032.032} C_VEL
LIN {X 0,Y 439.389,Z 351.754,A -85,B 0,C 180,E1 -9035.342,E2 -9035.342} C_VEL
LIN {X 0,Y 439.393,Z 351.75,A -85,B 0,C 180,E1 -9038.594,E2 -9038.594} C_VEL
LIN {X 0,Y 439.399,Z 351.754,A -85,B 0,C 180,E1 -9041.26,E2 -9041.26} C_VEL
LIN {X 0,Y 439.405,Z 351.75,A -85,B 0,C 180,E1 -9044.729,E2 -9044.729} C_VEL
LIN {X 0,Y 439.407,Z 351.748,A -85,B 0,C 180,E1 -9047.799,E2 -9047.799} C_VEL
LIN {X 0,Y 439.448,Z 351.743,A -85,B 0,C 180,E1 -9050.231,E2 -9050.231} C_VEL
LIN {X 0,Y 439.374,Z 351.752,A -85,B 0,C 180,E1 -9053.715,E2 -9053.715} C_VEL
LIN {X 0,Y 439.373,Z 351.758,A -85,B 0,C 180,E1 -9057.056,E2 -9057.056} C_VEL
LIN {X 0,Y 439.442,Z 351.751,A -85,B 0,C 180,E1 -9060.806,E2 -9060.806} C_VEL
LIN {X 0,Y 439.494,Z 351.94,A -85,B 0,C 180,E1 -9061.138,E2 -9061.138} C_VEL
LIN {X 0,Y 442.584,Z 366.648,A -85,B 0,C 180,E1 -9063.856,E2 -9063.856} C_VEL
LIN {X 0,Y 442.761,Z 371.067,A -85,B 0,C 180,E1 -9064.624,E2 -9064.624} C_VEL
LIN {X 0,Y 441.662,Z 390.01,A -85,B 0,C 180,E1 -9067.796,E2 -9067.796} C_VEL
LIN {X 0,Y 440.633,Z 410.338,A -85,B 0,C 180,E1 -9071.158,E2 -9071.158} C_VEL
LIN {X 0,Y 440.406,Z 415.459,A -85,B 0,C 180,E1 -9072,E2 -9072} C_VEL
LIN {X 0,Y 443.527,Z 440.079,A -85,B 0,C 180,E1 -9072.611,E2 -9072.611} C_VEL
LIN {X 0,Y 442.338,Z 525.51,A -85,B 0,C 180,E1 -9074.242,E2 -9074.242} C_VEL
LIN {X 0,Y 441.815,Z 539.382,A -85,B 0,C 180,E1 -9074.696,E2 -9074.696} C_VEL
LIN {X 0,Y 441.309,Z 551.894,A -85,B 0,C 180,E1 -9075.298,E2 -9075.298} C_VEL
LIN {X 0,Y 440.76,Z 563.557,A -85,B 0,C 180,E1 -9076.046,E2 -9076.046} C_VEL
LIN {X 0,Y 440.155,Z 574.215,A -85,B 0,C 180,E1 -9076.905,E2 -9076.905} C_VEL
LIN {X 0,Y 439.71,Z 584.13,A -85,B 0,C 180,E1 -9077.892,E2 -9077.892} C_VEL
LIN {X 0,Y 439.344,Z 592.757,A -85,B 0,C 180,E1 -9078.934,E2 -9078.934} C_VEL
LIN {X 0,Y 438.919,Z 602.085,A -85,B 0,C 180,E1 -9080.322,E2 -9080.322} C_VEL
LIN {X 0,Y 438.665,Z 609.591,A -85,B 0,C 180,E1 -9081.711,E2 -9081.711} C_VEL
LIN {X 0,Y 438.52,Z 615.584,A -85,B 0,C 180,E1 -9083.098,E2 -9083.098} C_VEL
LIN {X 0,Y 438.465,Z 620.266,A -85,B 0,C 180,E1 -9084.482,E2 -9084.482} C_VEL
LIN {X 0,Y 438.391,Z 623.784,A -85,B 0,C 180,E1 -9085.864,E2 -9085.864} C_VEL
LIN {X 0,Y 438.458,Z 626.251,A -85,B 0,C 180,E1 -9087.245,E2 -9087.245} C_VEL
LIN {X 0,Y 438.461,Z 627.311,A -85,B 0,C 180,E1 -9088.164,E2 -9088.164} C_VEL
LIN {X 0,Y 438.38,Z 627.941,A -85,B 0,C 180,E1 -9089.082,E2 -9089.082} C_VEL
LIN {X 0,Y 438.363,Z 628.162,A -85,B 0,C 180,E1 -9090.001,E2 -9090.001} C_VEL
LIN {X 0,Y 438.382,Z 627.944,A -85,B 0,C 180,E1 -9090.92,E2 -9090.92} C_VEL
LIN {X 0,Y 438.464,Z 627.273,A -85,B 0,C 180,E1 -9091.838,E2 -9091.838} C_VEL
LIN {X 0,Y 438.477,Z 626.182,A -85,B 0,C 180,E1 -9092.757,E2 -9092.757} C_VEL
LIN {X 0,Y 438.406,Z 623.701,A -85,B 0,C 180,E1 -9094.138,E2 -9094.138} C_VEL
LIN {X 0,Y 438.453,Z 620.171,A -85,B 0,C 180,E1 -9095.52,E2 -9095.52} C_VEL
LIN {X 0,Y 438.56,Z 614.716,A -85,B 0,C 180,E1 -9097.112,E2 -9097.112} C_VEL
LIN {X 0,Y 438.683,Z 608.434,A -85,B 0,C 180,E1 -9098.523,E2 -9098.523} C_VEL
LIN {X 0,Y 438.929,Z 600.731,A -85,B 0,C 180,E1 -9099.912,E2 -9099.912} C_VEL
LIN {X 0,Y 439.411,Z 591.2,A -85,B 0,C 180,E1 -9101.3,E2 -9101.3} C_VEL
LIN {X 0,Y 439.876,Z 582.425,A -85,B 0,C 180,E1 -9102.34,E2 -9102.34} C_VEL
LIN {X 0,Y 440.463,Z 570.424,A -85,B 0,C 180,E1 -9103.496,E2 -9103.496} C_VEL
LIN {X 0,Y 441.121,Z 558.329,A -85,B 0,C 180,E1 -9104.416,E2 -9104.416} C_VEL
LIN {X 0,Y 441.787,Z 545.553,A -85,B 0,C 180,E1 -9105.159,E2 -9105.159} C_VEL
LIN {X 0,Y 442.393,Z 532.286,A -85,B 0,C 180,E1 -9105.728,E2 -9105.728} C_VEL
LIN {X 0,Y 442.889,Z 518.026,A -85,B 0,C 180,E1 -9106.124,E2 -9106.124} C_VEL
LIN {X 0,Y 444.224,Z 439.866,A -85,B 0,C 180,E1 -9107.7,E2 -9107.7} C_VEL
LIN {X 0,Y 441.506,Z 418.003,A -85,B 0,C 180,E1 -9108.328,E2 -9108.328} C_VEL
LIN {X 0,Y 440.472,Z 411.385,A -85,B 0,C 180,E1 -9108.552,E2 -9108.552} C_VEL
LIN {X 0,Y 441.428,Z 394.137,A -85,B 0,C 180,E1 -9111.481,E2 -9111.481} C_VEL
LIN {X 0,Y 442.821,Z 373.633,A -85,B 0,C 180,E1 -9115.084,E2 -9115.084} C_VEL
LIN {X 0,Y 443.117,Z 369.343,A -85,B 0,C 180,E1 -9115.86,E2 -9115.86} C_VEL
LIN {X 0,Y 441.752,Z 361.404,A -85,B 0,C 180,E1 -9117.477,E2 -9117.477} C_VEL
LIN {X 0,Y 439.425,Z 351.752,A -85,B 0,C 180,E1 -9119.658,E2 -9119.658} C_VEL
LIN {X 0,Y 439.378,Z 351.758,A -85,B 0,C 180,E1 -9122.946,E2 -9122.946} C_VEL
LIN {X 0,Y 439.379,Z 351.755,A -85,B 0,C 180,E1 -9126.288,E2 -9126.288} C_VEL
LIN {X 0,Y 439.412,Z 351.75,A -85,B 0,C 180,E1 -9129.85,E2 -9129.85} C_VEL
LIN {X 0,Y 439.388,Z 351.753,A -85,B 0,C 180,E1 -9132.627,E2 -9132.627} C_VEL
LIN {X 0,Y 439.407,Z 351.752,A -85,B 0,C 180,E1 -9135.271,E2 -9135.271} C_VEL
LIN {X 0,Y 439.394,Z 351.754,A -85,B 0,C 180,E1 -9138.744,E2 -9138.744} C_VEL
LIN {X 0,Y 439.382,Z 351.753,A -85,B 0,C 180,E1 -9141.608,E2 -9141.608} C_VEL
LIN {X 0,Y 439.404,Z 351.753,A -85,B 0,C 180,E1 -9144.844,E2 -9144.844} C_VEL
LIN {X 0,Y 439.378,Z 351.754,A -85,B 0,C 180,E1 -9148.14,E2 -9148.14} C_VEL
LIN {X 0,Y 439.438,Z 351.746,A -85,B 0,C 180,E1 -9151.598,E2 -9151.598} C_VEL
LIN {X 0,Y 439.411,Z 351.752,A -85,B 0,C 180,E1 -9154.415,E2 -9154.415} C_VEL
LIN {X 0,Y 439.37,Z 351.757,A -85,B 0,C 180,E1 -9157.425,E2 -9157.425} C_VEL
LIN {X 0,Y 439.449,Z 351.901,A -85,B 0,C 180,E1 -9159.95,E2 -9159.95} C_VEL
LIN {X 0,Y 440.593,Z 357.079,A -85,B 0,C 180,E1 -9161.566,E2 -9161.566} C_VEL
LIN {X 0,Y 445.096,Z 368.665,A -85,B 0,C 180,E1 -9162.104,E2 -9162.104} C_VEL
LIN {X 0,Y 443.469,Z 450.633,A -85,B 0,C 180,E1 -9163.81,E2 -9163.81} C_VEL
LIN {X 0,Y 443.193,Z 465.478,A -85,B 0,C 180,E1 -9164.154,E2 -9164.154} C_VEL
LIN {X 0,Y 442.855,Z 478.489,A -85,B 0,C 180,E1 -9164.643,E2 -9164.643} C_VEL
LIN {X 0,Y 442.392,Z 491.529,A -85,B 0,C 180,E1 -9165.337,E2 -9165.337} C_VEL
LIN {X 0,Y 441.903,Z 503.644,A -85,B 0,C 180,E1 -9166.198,E2 -9166.198} C_VEL
LIN {X 0,Y 441.261,Z 515.088,A -85,B 0,C 180,E1 -9167.233,E2 -9167.233} C_VEL
LIN {X 0,Y 440.718,Z 524.338,A -85,B 0,C 180,E1 -9168.269,E2 -9168.269} C_VEL
LIN {X 0,Y 440.305,Z 532.726,A -85,B 0,C 180,E1 -9169.423,E2 -9169.423} C_VEL
LIN {X 0,Y 439.829,Z 540.889,A -85,B 0,C 180,E1 -9170.805,E2 -9170.805} C_VEL
LIN {X 0,Y 439.378,Z 547.451,A -85,B 0,C 180,E1 -9172.186,E2 -9172.186} C_VEL
LIN {X 0,Y 438.98,Z 552.645,A -85,B 0,C 180,E1 -9173.565,E2 -9173.565} C_VEL
LIN {X 0,Y 438.933,Z 556.611,A -85,B 0,C 180,E1 -9174.948,E2 -9174.948} C_VEL
LIN {X 0,Y 438.836,Z 559.508,A -85,B 0,C 180,E1 -9176.327,E2 -9176.327} C_VEL
LIN {X 0,Y 438.652,Z 560.878,A -85,B 0,C 180,E1 -9177.245,E2 -9177.245} C_VEL
LIN {X 0,Y 438.488,Z 561.827,A -85,B 0,C 180,E1 -9178.163,E2 -9178.163} C_VEL
LIN {X 0,Y 438.404,Z 562.371,A -85,B 0,C 180,E1 -9179.081,E2 -9179.081} C_VEL
LIN {X 0,Y 438.382,Z 562.489,A -85,B 0,C 180,E1 -9180,E2 -9180} C_VEL
LIN {X 0,Y 438.402,Z 562.158,A -85,B 0,C 180,E1 -9180.918,E2 -9180.918} C_VEL
LIN {X 0,Y 438.484,Z 561.423,A -85,B 0,C 180,E1 -9181.837,E2 -9181.837} C_VEL
LIN {X 0,Y 438.622,Z 560.285,A -85,B 0,C 180,E1 -9182.755,E2 -9182.755} C_VEL
LIN {X 0,Y 438.727,Z 557.743,A -85,B 0,C 180,E1 -9184.134,E2 -9184.134} C_VEL
LIN {X 0,Y 438.73,Z 554.18,A -85,B 0,C 180,E1 -9185.515,E2 -9185.515} C_VEL
LIN {X 0,Y 439.045,Z 548.922,A -85,B 0,C 180,E1 -9187.035,E2 -9187.035} C_VEL
LIN {X 0,Y 439.3,Z 542.339,A -85,B 0,C 180,E1 -9188.51,E2 -9188.51} C_VEL
LIN {X 0,Y 439.702,Z 534.6,A -85,B 0,C 180,E1 -9189.894,E2 -9189.894} C_VEL
LIN {X 0,Y 440.106,Z 526.678,A -85,B 0,C 180,E1 -9191.048,E2 -9191.048} C_VEL
LIN {X 0,Y 440.647,Z 515.895,A -85,B 0,C 180,E1 -9192.317,E2 -9192.317} C_VEL
LIN {X 0,Y 441.214,Z 504.654,A -85,B 0,C 180,E1 -9193.375,E2 -9193.375} C_VEL
LIN {X 0,Y 441.612,Z 492.403,A -85,B 0,C 180,E1 -9194.281,E2 -9194.281} C_VEL
LIN {X 0,Y 442.051,Z 480.239,A -85,B 0,C 180,E1 -9194.972,E2 -9194.972} C_VEL
LIN {X 0,Y 442.386,Z 466.809,A -85,B 0,C 180,E1 -9195.521,E2 -9195.521} C_VEL
LIN {X 0,Y 442.683,Z 453.773,A -85,B 0,C 180,E1 -9195.864,E2 -9195.864} C_VEL
LIN {X 0,Y 443.851,Z 367.404,A -85,B 0,C 180,E1 -9197.494,E2 -9197.494} C_VEL
LIN {X 0,Y 440.543,Z 355.555,A -85,B 0,C 180,E1 -9197.851,E2 -9197.851} C_VEL
LIN {X 0,Y 439.471,Z 351.935,A -85,B 0,C 180,E1 -9197.982,E2 -9197.982} C_VEL
LIN {X 0,Y 439.393,Z 351.752,A -85,B 0,C 180,E1 -9200.603,E2 -9200.603} C_VEL
LIN {X 0,Y 439.417,Z 351.748,A -85,B 0,C 180,E1 -9204.264,E2 -9204.264} C_VEL
LIN {X 0,Y 439.445,Z 351.746,A -85,B 0,C 180,E1 -9207.632,E2 -9207.632} C_VEL
LIN {X 0,Y 439.366,Z 351.758,A -85,B 0,C 180,E1 -9210.788,E2 -9210.788} C_VEL
LIN {X 0,Y 439.392,Z 351.752,A -85,B 0,C 180,E1 -9214.043,E2 -9214.043} C_VEL
LIN {X 0,Y 439.353,Z 351.759,A -85,B 0,C 180,E1 -9216.887,E2 -9216.887} C_VEL
LIN {X 0,Y 439.411,Z 351.75,A -85,B 0,C 180,E1 -9219.849,E2 -9219.849} C_VEL
LIN {X 0,Y 439.387,Z 351.755,A -85,B 0,C 180,E1 -9222.627,E2 -9222.627} C_VEL
LIN {X 0,Y 439.406,Z 351.751,A -85,B 0,C 180,E1 -9225.27,E2 -9225.27} C_VEL
LIN {X 0,Y 439.393,Z 351.754,A -85,B 0,C 180,E1 -9228.743,E2 -9228.743} C_VEL
LIN {X 0,Y 439.381,Z 351.754,A -85,B 0,C 180,E1 -9231.607,E2 -9231.607} C_VEL
LIN {X 0,Y 439.404,Z 351.752,A -85,B 0,C 180,E1 -9234.843,E2 -9234.843} C_VEL
LIN {X 0,Y 439.377,Z 351.754,A -85,B 0,C 180,E1 -9238.139,E2 -9238.139} C_VEL
LIN {X 0,Y 439.436,Z 351.746,A -85,B 0,C 180,E1 -9241.597,E2 -9241.597} C_VEL
LIN {X 0,Y 439.41,Z 351.752,A -85,B 0,C 180,E1 -9244.414,E2 -9244.414} C_VEL
LIN {X 0,Y 439.369,Z 351.755,A -85,B 0,C 180,E1 -9247.424,E2 -9247.424} C_VEL
LIN {X 0,Y 439.445,Z 351.747,A -85,B 0,C 180,E1 -9250.662,E2 -9250.662} C_VEL
LIN {X 0,Y 439.466,Z 351.744,A -85,B 0,C 180,E1 -9254.224,E2 -9254.224} C_VEL
LIN {X 0,Y 439.421,Z 351.747,A -85,B 0,C 180,E1 -9255.866,E2 -9255.866} C_VEL
LIN {X 0,Y 438.765,Z 351.833,A -85,B 0,C 180,E1 -9256.631,E2 -9256.631} C_VEL
LIN {X 0,Y 435.922,Z 352.187,A -85,B 0,C 180,E1 -9257.874,E2 -9257.874} C_VEL
LIN {X 0,Y 433.517,Z 352.485,A -85,B 0,C 180,E1 -9258.877,E2 -9258.877} C_VEL
LIN {X 0,Y 432.489,Z 352.611,A -85,B 0,C 180,E1 -9259.652,E2 -9259.652} C_VEL
LIN {X 0,Y 432.409,Z 352.62,A -85,B 0,C 180,E1 -9259.914,E2 -9259.914} C_VEL
LIN {X 0,Y 432.556,Z 352.605,A -85,B 0,C 180,E1 -9262.53,E2 -9262.53} C_VEL
LIN {X 0,Y 432.597,Z 352.601,A -85,B 0,C 180,E1 -9264.405,E2 -9264.405} C_VEL
LIN {X 0,Y 432.609,Z 352.599,A -85,B 0,C 180,E1 -9268.137,E2 -9268.137} C_VEL
LIN {X 0,Y 432.736,Z 352.582,A -85,B 0,C 180,E1 -9269.999,E2 -9269.999} C_VEL
LIN {X 0,Y 432.607,Z 352.597,A -85,B 0,C 180,E1 -9272.792,E2 -9272.792} C_VEL
LIN {X 0,Y 432.575,Z 352.602,A -85,B 0,C 180,E1 -9276.529,E2 -9276.529} C_VEL
LIN {X 0,Y 432.444,Z 352.616,A -85,B 0,C 180,E1 -9279.352,E2 -9279.352} C_VEL
LIN {X 0,Y 432.43,Z 352.618,A -85,B 0,C 180,E1 -9282.802,E2 -9282.802} C_VEL
LIN {X 0,Y 432.422,Z 352.621,A -85,B 0,C 180,E1 -9286.483,E2 -9286.483} C_VEL
LIN {X 0,Y 432.338,Z 352.633,A -85,B 0,C 180,E1 -9289.959,E2 -9289.959} C_VEL
LIN {X 0,Y 432.317,Z 352.632,A -85,B 0,C 180,E1 -9292.963,E2 -9292.963} C_VEL
LIN {X 0,Y 432.362,Z 352.631,A -85,B 0,C 180,E1 -9296.031,E2 -9296.031} C_VEL
LIN {X 0,Y 432.349,Z 352.628,A -85,B 0,C 180,E1 -9299.185,E2 -9299.185} C_VEL
LIN {X 0,Y 432.327,Z 352.633,A -85,B 0,C 180,E1 -9302.294,E2 -9302.294} C_VEL
LIN {X 0,Y 432.336,Z 352.629,A -85,B 0,C 180,E1 -9304.676,E2 -9304.676} C_VEL
LIN {X 0,Y 432.349,Z 352.631,A -85,B 0,C 180,E1 -9308.147,E2 -9308.147} C_VEL
LIN {X 0,Y 432.367,Z 352.627,A -85,B 0,C 180,E1 -9311.607,E2 -9311.607} C_VEL
LIN {X 0,Y 432.372,Z 352.626,A -85,B 0,C 180,E1 -9314.34,E2 -9314.34} C_VEL
LIN {X 0,Y 432.359,Z 352.626,A -85,B 0,C 180,E1 -9317.008,E2 -9317.008} C_VEL
LIN {X 0,Y 432.353,Z 352.632,A -85,B 0,C 180,E1 -9319.815,E2 -9319.815} C_VEL
LIN {X 0,Y 432.31,Z 352.632,A -85,B 0,C 180,E1 -9323.022,E2 -9323.022} C_VEL
LIN {X 0,Y 432.351,Z 352.631,A -85,B 0,C 180,E1 -9325.996,E2 -9325.996} C_VEL
LIN {X 0,Y 432.386,Z 352.628,A -85,B 0,C 180,E1 -9329.743,E2 -9329.743} C_VEL
LIN {X 0,Y 432.391,Z 352.624,A -85,B 0,C 180,E1 -9333.372,E2 -9333.372} C_VEL
LIN {X 0,Y 432.362,Z 352.628,A -85,B 0,C 180,E1 -9336.023,E2 -9336.023} C_VEL
LIN {X 0,Y 432.341,Z 352.628,A -85,B 0,C 180,E1 -9339.046,E2 -9339.046} C_VEL
LIN {X 0,Y 432.369,Z 352.627,A -85,B 0,C 180,E1 -9342.011,E2 -9342.011} C_VEL
LIN {X 0,Y 432.392,Z 352.621,A -85,B 0,C 180,E1 -9344.926,E2 -9344.926} C_VEL
LIN {X 0,Y 432.471,Z 352.616,A -85,B 0,C 180,E1 -9347.804,E2 -9347.804} C_VEL
LIN {X 0,Y 432.482,Z 352.617,A -85,B 0,C 180,E1 -9351.59,E2 -9351.59} C_VEL
LIN {X 0,Y 432.589,Z 352.596,A -85,B 0,C 180,E1 -9354.406,E2 -9354.406} C_VEL
LIN {X 0,Y 432.596,Z 352.596,A -85,B 0,C 180,E1 -9358.138,E2 -9358.138} C_VEL
LIN {X 0,Y 432.725,Z 352.581,A -85,B 0,C 180,E1 -9360,E2 -9360} C_VEL
LIN {X 0,Y 432.597,Z 352.595,A -85,B 0,C 180,E1 -9362.794,E2 -9362.794} C_VEL
LIN {X 0,Y 432.566,Z 352.598,A -85,B 0,C 180,E1 -9366.531,E2 -9366.531} C_VEL
LIN {X 0,Y 432.435,Z 352.621,A -85,B 0,C 180,E1 -9369.353,E2 -9369.353} C_VEL
LIN {X 0,Y 432.435,Z 352.616,A -85,B 0,C 180,E1 -9372.812,E2 -9372.812} C_VEL
LIN {X 0,Y 432.403,Z 352.619,A -85,B 0,C 180,E1 -9376.48,E2 -9376.48} C_VEL
LIN {X 0,Y 432.33,Z 352.629,A -85,B 0,C 180,E1 -9379.961,E2 -9379.961} C_VEL
LIN {X 0,Y 432.311,Z 352.634,A -85,B 0,C 180,E1 -9382.965,E2 -9382.965} C_VEL
LIN {X 0,Y 432.356,Z 352.626,A -85,B 0,C 180,E1 -9386.033,E2 -9386.033} C_VEL
LIN {X 0,Y 432.335,Z 352.634,A -85,B 0,C 180,E1 -9389.188,E2 -9389.188} C_VEL
LIN {X 0,Y 432.315,Z 352.631,A -85,B 0,C 180,E1 -9392.444,E2 -9392.444} C_VEL
LIN {X 0,Y 432.339,Z 352.63,A -85,B 0,C 180,E1 -9395.633,E2 -9395.633} C_VEL
LIN {X 0,Y 432.354,Z 352.628,A -85,B 0,C 180,E1 -9398.719,E2 -9398.719} C_VEL
LIN {X 0,Y 432.368,Z 352.625,A -85,B 0,C 180,E1 -9401.793,E2 -9401.793} C_VEL
LIN {X 0,Y 432.372,Z 352.624,A -85,B 0,C 180,E1 -9404.343,E2 -9404.343} C_VEL
LIN {X 0,Y 432.361,Z 352.63,A -85,B 0,C 180,E1 -9407.01,E2 -9407.01} C_VEL
LIN {X 0,Y 432.354,Z 352.627,A -85,B 0,C 180,E1 -9409.818,E2 -9409.818} C_VEL
LIN {X 0,Y 432.314,Z 352.637,A -85,B 0,C 180,E1 -9413.024,E2 -9413.024} C_VEL
LIN {X 0,Y 432.356,Z 352.626,A -85,B 0,C 180,E1 -9415.998,E2 -9415.998} C_VEL
LIN {X 0,Y 432.394,Z 352.626,A -85,B 0,C 180,E1 -9419.746,E2 -9419.746} C_VEL
LIN {X 0,Y 432.418,Z 352.682,A -85,B 0,C 180,E1 -9420.891,E2 -9420.891} C_VEL
LIN {X 0,Y 435.551,Z 367.403,A -85,B 0,C 180,E1 -9423.659,E2 -9423.659} C_VEL
LIN {X 0,Y 435.83,Z 371.85,A -85,B 0,C 180,E1 -9424.447,E2 -9424.447} C_VEL
LIN {X 0,Y 434.583,Z 392.227,A -85,B 0,C 180,E1 -9427.916,E2 -9427.916} C_VEL
LIN {X 0,Y 433.484,Z 413.985,A -85,B 0,C 180,E1 -9431.571,E2 -9431.571} C_VEL
LIN {X 0,Y 433.421,Z 415.163,A -85,B 0,C 180,E1 -9431.767,E2 -9431.767} C_VEL
LIN {X 0,Y 436.655,Z 441.422,A -85,B 0,C 180,E1 -9432.41,E2 -9432.41} C_VEL
LIN {X 0,Y 435.413,Z 524.916,A -85,B 0,C 180,E1 -9434.045,E2 -9434.045} C_VEL
LIN {X 0,Y 434.858,Z 538.768,A -85,B 0,C 180,E1 -9434.505,E2 -9434.505} C_VEL
LIN {X 0,Y 434.347,Z 551.311,A -85,B 0,C 180,E1 -9435.117,E2 -9435.117} C_VEL
LIN {X 0,Y 433.741,Z 563.78,A -85,B 0,C 180,E1 -9435.935,E2 -9435.935} C_VEL
LIN {X 0,Y 433.093,Z 574.993,A -85,B 0,C 180,E1 -9436.87,E2 -9436.87} C_VEL
LIN {X 0,Y 432.656,Z 584.123,A -85,B 0,C 180,E1 -9437.81,E2 -9437.81} C_VEL
LIN {X 0,Y 432.245,Z 593.499,A -85,B 0,C 180,E1 -9438.987,E2 -9438.987} C_VEL
LIN {X 0,Y 431.814,Z 602.618,A -85,B 0,C 180,E1 -9440.398,E2 -9440.398} C_VEL
LIN {X 0,Y 431.578,Z 609.927,A -85,B 0,C 180,E1 -9441.809,E2 -9441.809} C_VEL
LIN {X 0,Y 431.437,Z 616.553,A -85,B 0,C 180,E1 -9443.454,E2 -9443.454} C_VEL
LIN {X 0,Y 431.375,Z 620.884,A -85,B 0,C 180,E1 -9444.86,E2 -9444.86} C_VEL
LIN {X 0,Y 431.362,Z 624.082,A -85,B 0,C 180,E1 -9446.264,E2 -9446.264} C_VEL
LIN {X 0,Y 431.384,Z 625.652,A -85,B 0,C 180,E1 -9447.2,E2 -9447.2} C_VEL
LIN {X 0,Y 431.404,Z 626.737,A -85,B 0,C 180,E1 -9448.134,E2 -9448.134} C_VEL
LIN {X 0,Y 431.321,Z 627.379,A -85,B 0,C 180,E1 -9449.067,E2 -9449.067} C_VEL
LIN {X 0,Y 431.301,Z 627.61,A -85,B 0,C 180,E1 -9450.001,E2 -9450.001} C_VEL
LIN {X 0,Y 431.323,Z 627.412,A -85,B 0,C 180,E1 -9450.935,E2 -9450.935} C_VEL
LIN {X 0,Y 431.391,Z 626.75,A -85,B 0,C 180,E1 -9451.868,E2 -9451.868} C_VEL
LIN {X 0,Y 431.403,Z 625.662,A -85,B 0,C 180,E1 -9452.802,E2 -9452.802} C_VEL
LIN {X 0,Y 431.312,Z 623.185,A -85,B 0,C 180,E1 -9454.206,E2 -9454.206} C_VEL
LIN {X 0,Y 431.353,Z 619.665,A -85,B 0,C 180,E1 -9455.611,E2 -9455.611} C_VEL
LIN {X 0,Y 431.472,Z 615.007,A -85,B 0,C 180,E1 -9457.018,E2 -9457.018} C_VEL
LIN {X 0,Y 431.599,Z 609.078,A -85,B 0,C 180,E1 -9458.428,E2 -9458.428} C_VEL
LIN {X 0,Y 431.829,Z 601.688,A -85,B 0,C 180,E1 -9459.84,E2 -9459.84} C_VEL
LIN {X 0,Y 432.31,Z 592.473,A -85,B 0,C 180,E1 -9461.251,E2 -9461.251} C_VEL
LIN {X 0,Y 432.735,Z 584.077,A -85,B 0,C 180,E1 -9462.309,E2 -9462.309} C_VEL
LIN {X 0,Y 433.334,Z 573.11,A -85,B 0,C 180,E1 -9463.447,E2 -9463.447} C_VEL
LIN {X 0,Y 434.068,Z 561.351,A -85,B 0,C 180,E1 -9464.416,E2 -9464.416} C_VEL
LIN {X 0,Y 434.764,Z 548.762,A -85,B 0,C 180,E1 -9465.23,E2 -9465.23} C_VEL
LIN {X 0,Y 435.41,Z 535.479,A -85,B 0,C 180,E1 -9465.867,E2 -9465.867} C_VEL
LIN {X 0,Y 436.084,Z 521.497,A -85,B 0,C 180,E1 -9466.322,E2 -9466.322} C_VEL
LIN {X 0,Y 437.586,Z 440.561,A -85,B 0,C 180,E1 -9468.021,E2 -9468.021} C_VEL
LIN {X 0,Y 435.068,Z 419.666,A -85,B 0,C 180,E1 -9468.643,E2 -9468.643} C_VEL
LIN {X 0,Y 433.604,Z 410.524,A -85,B 0,C 180,E1 -9468.977,E2 -9468.977} C_VEL
LIN {X 0,Y 434.734,Z 391.313,A -85,B 0,C 180,E1 -9472.329,E2 -9472.329} C_VEL
LIN {X 0,Y 436.277,Z 372.234,A -85,B 0,C 180,E1 -9475.783,E2 -9475.783} C_VEL
LIN {X 0,Y 435.733,Z 366.937,A -85,B 0,C 180,E1 -9476.848,E2 -9476.848} C_VEL
LIN {X 0,Y 433.431,Z 356.754,A -85,B 0,C 180,E1 -9479.108,E2 -9479.108} C_VEL
LIN {X 0,Y 432.342,Z 352.633,A -85,B 0,C 180,E1 -9480.126,E2 -9480.126} C_VEL
LIN {X 0,Y 432.345,Z 352.634,A -85,B 0,C 180,E1 -9483.553,E2 -9483.553} C_VEL
LIN {X 0,Y 432.343,Z 352.632,A -85,B 0,C 180,E1 -9485.818,E2 -9485.818} C_VEL
LIN {X 0,Y 432.356,Z 352.63,A -85,B 0,C 180,E1 -9489.343,E2 -9489.343} C_VEL
LIN {X 0,Y 432.339,Z 352.63,A -85,B 0,C 180,E1 -9491.797,E2 -9491.797} C_VEL
LIN {X 0,Y 432.339,Z 352.631,A -85,B 0,C 180,E1 -9494.348,E2 -9494.348} C_VEL
LIN {X 0,Y 432.326,Z 352.635,A -85,B 0,C 180,E1 -9497.016,E2 -9497.016} C_VEL
LIN {X 0,Y 432.342,Z 352.63,A -85,B 0,C 180,E1 -9499.821,E2 -9499.821} C_VEL
LIN {X 0,Y 432.312,Z 352.636,A -85,B 0,C 180,E1 -9503.022,E2 -9503.022} C_VEL
LIN {X 0,Y 432.365,Z 352.626,A -85,B 0,C 180,E1 -9505.997,E2 -9505.997} C_VEL
LIN {X 0,Y 432.353,Z 352.629,A -85,B 0,C 180,E1 -9509.49,E2 -9509.49} C_VEL
LIN {X 0,Y 432.397,Z 352.626,A -85,B 0,C 180,E1 -9512.928,E2 -9512.928} C_VEL
LIN {X 0,Y 432.377,Z 352.627,A -85,B 0,C 180,E1 -9516.024,E2 -9516.024} C_VEL
LIN {X 0,Y 432.384,Z 352.768,A -85,B 0,C 180,E1 -9519.483,E2 -9519.483} C_VEL
LIN {X 0,Y 433.54,Z 357.904,A -85,B 0,C 180,E1 -9521.146,E2 -9521.146} C_VEL
LIN {X 0,Y 438.462,Z 370,A -85,B 0,C 180,E1 -9521.753,E2 -9521.753} C_VEL
LIN {X 0,Y 438.52,Z 373.878,A -85,B 0,C 180,E1 -9521.849,E2 -9521.849} C_VEL
LIN {X 0,Y 436.684,Z 453.534,A -85,B 0,C 180,E1 -9523.551,E2 -9523.551} C_VEL
LIN {X 0,Y 436.49,Z 467.451,A -85,B 0,C 180,E1 -9523.904,E2 -9523.904} C_VEL
LIN {X 0,Y 436.051,Z 481.159,A -85,B 0,C 180,E1 -9524.457,E2 -9524.457} C_VEL
LIN {X 0,Y 435.585,Z 493.703,A -85,B 0,C 180,E1 -9525.167,E2 -9525.167} C_VEL
LIN {X 0,Y 434.992,Z 506.072,A -85,B 0,C 180,E1 -9526.094,E2 -9526.094} C_VEL
LIN {X 0,Y 434.356,Z 517.155,A -85,B 0,C 180,E1 -9527.145,E2 -9527.145} C_VEL
LIN {X 0,Y 433.717,Z 526.981,A -85,B 0,C 180,E1 -9528.314,E2 -9528.314} C_VEL
LIN {X 0,Y 433.279,Z 535.012,A -85,B 0,C 180,E1 -9529.486,E2 -9529.486} C_VEL
LIN {X 0,Y 432.776,Z 542.887,A -85,B 0,C 180,E1 -9530.89,E2 -9530.89} C_VEL
LIN {X 0,Y 432.399,Z 548.194,A -85,B 0,C 180,E1 -9532.059,E2 -9532.059} C_VEL
LIN {X 0,Y 431.96,Z 553.351,A -85,B 0,C 180,E1 -9533.46,E2 -9533.46} C_VEL
LIN {X 0,Y 431.903,Z 557.281,A -85,B 0,C 180,E1 -9534.865,E2 -9534.865} C_VEL
LIN {X 0,Y 431.796,Z 560.15,A -85,B 0,C 180,E1 -9536.267,E2 -9536.267} C_VEL
LIN {X 0,Y 431.608,Z 561.497,A -85,B 0,C 180,E1 -9537.2,E2 -9537.2} C_VEL
LIN {X 0,Y 431.435,Z 562.429,A -85,B 0,C 180,E1 -9538.133,E2 -9538.133} C_VEL
LIN {X 0,Y 431.344,Z 562.953,A -85,B 0,C 180,E1 -9539.066,E2 -9539.066} C_VEL
LIN {X 0,Y 431.32,Z 563.036,A -85,B 0,C 180,E1 -9540,E2 -9540} C_VEL
LIN {X 0,Y 431.342,Z 562.681,A -85,B 0,C 180,E1 -9540.933,E2 -9540.933} C_VEL
LIN {X 0,Y 431.431,Z 561.923,A -85,B 0,C 180,E1 -9541.867,E2 -9541.867} C_VEL
LIN {X 0,Y 431.545,Z 560.756,A -85,B 0,C 180,E1 -9542.8,E2 -9542.8} C_VEL
LIN {X 0,Y 431.67,Z 558.167,A -85,B 0,C 180,E1 -9544.201,E2 -9544.201} C_VEL
LIN {X 0,Y 431.678,Z 554.548,A -85,B 0,C 180,E1 -9545.606,E2 -9545.606} C_VEL
LIN {X 0,Y 431.992,Z 549.55,A -85,B 0,C 180,E1 -9547.065,E2 -9547.065} C_VEL
LIN {X 0,Y 432.262,Z 542.551,A -85,B 0,C 180,E1 -9548.65,E2 -9548.65} C_VEL
LIN {X 0,Y 432.686,Z 534.725,A -85,B 0,C 180,E1 -9550.056,E2 -9550.056} C_VEL
LIN {X 0,Y 433.103,Z 526.686,A -85,B 0,C 180,E1 -9551.229,E2 -9551.229} C_VEL
LIN {X 0,Y 433.636,Z 516.865,A -85,B 0,C 180,E1 -9552.4,E2 -9552.4} C_VEL
LIN {X 0,Y 434.161,Z 506.414,A -85,B 0,C 180,E1 -9553.416,E2 -9553.416} C_VEL
LIN {X 0,Y 434.538,Z 495.414,A -85,B 0,C 180,E1 -9554.279,E2 -9554.279} C_VEL
LIN {X 0,Y 435.014,Z 482.809,A -85,B 0,C 180,E1 -9555.04,E2 -9555.04} C_VEL
LIN {X 0,Y 435.466,Z 469.697,A -85,B 0,C 180,E1 -9555.624,E2 -9555.624} C_VEL
LIN {X 0,Y 435.735,Z 456.747,A -85,B 0,C 180,E1 -9556.004,E2 -9556.004} C_VEL
LIN {X 0,Y 436.922,Z 367.937,A -85,B 0,C 180,E1 -9557.73,E2 -9557.73} C_VEL
LIN {X 0,Y 432.422,Z 352.621,A -85,B 0,C 180,E1 -9558.232,E2 -9558.232} C_VEL
LIN {X 0,Y 432.362,Z 352.628,A -85,B 0,C 180,E1 -9561.954,E2 -9561.954} C_VEL
LIN {X 0,Y 432.353,Z 352.63,A -85,B 0,C 180,E1 -9565.001,E2 -9565.001} C_VEL
LIN {X 0,Y 432.386,Z 352.624,A -85,B 0,C 180,E1 -9568.123,E2 -9568.123} C_VEL
LIN {X 0,Y 432.326,Z 352.632,A -85,B 0,C 180,E1 -9571.346,E2 -9571.346} C_VEL
LIN {X 0,Y 432.344,Z 352.632,A -85,B 0,C 180,E1 -9574.677,E2 -9574.677} C_VEL
LIN {X 0,Y 432.341,Z 352.63,A -85,B 0,C 180,E1 -9578.149,E2 -9578.149} C_VEL
LIN {X 0,Y 432.337,Z 352.632,A -85,B 0,C 180,E1 -9581.602,E2 -9581.602} C_VEL
LIN {X 0,Y 432.338,Z 352.631,A -85,B 0,C 180,E1 -9584.347,E2 -9584.347} C_VEL
LIN {X 0,Y 432.325,Z 352.633,A -85,B 0,C 180,E1 -9587.015,E2 -9587.015} C_VEL
LIN {X 0,Y 432.341,Z 352.63,A -85,B 0,C 180,E1 -9589.82,E2 -9589.82} C_VEL
LIN {X 0,Y 432.311,Z 352.634,A -85,B 0,C 180,E1 -9593.021,E2 -9593.021} C_VEL
LIN {X 0,Y 432.363,Z 352.627,A -85,B 0,C 180,E1 -9595.996,E2 -9595.996} C_VEL
LIN {X 0,Y 432.352,Z 352.63,A -85,B 0,C 180,E1 -9599.489,E2 -9599.489} C_VEL
LIN {X 0,Y 432.395,Z 352.624,A -85,B 0,C 180,E1 -9602.928,E2 -9602.928} C_VEL
LIN {X 0,Y 432.376,Z 352.626,A -85,B 0,C 180,E1 -9606.023,E2 -9606.023} C_VEL
LIN {X 0,Y 432.354,Z 352.628,A -85,B 0,C 180,E1 -9609.045,E2 -9609.045} C_VEL
LIN {X 0,Y 432.382,Z 352.625,A -85,B 0,C 180,E1 -9612.01,E2 -9612.01} C_VEL
LIN {X 0,Y 432.399,Z 352.623,A -85,B 0,C 180,E1 -9614.926,E2 -9614.926} C_VEL
LIN {X 0,Y 432.462,Z 352.614,A -85,B 0,C 180,E1 -9617.803,E2 -9617.803} C_VEL
LIN {X 0,Y 432.409,Z 352.62,A -85,B 0,C 180,E1 -9619.914,E2 -9619.914} C_VEL
LIN {X 0,Y 431.758,Z 352.704,A -85,B 0,C 180,E1 -9620.693,E2 -9620.693} C_VEL
LIN {X 0,Y 428.95,Z 353.053,A -85,B 0,C 180,E1 -9621.959,E2 -9621.959} C_VEL
LIN {X 0,Y 426.588,Z 353.346,A -85,B 0,C 180,E1 -9622.981,E2 -9622.981} C_VEL
LIN {X 0,Y 425.6,Z 353.47,A -85,B 0,C 180,E1 -9623.77,E2 -9623.77} C_VEL
LIN {X 0,Y 425.533,Z 353.479,A -85,B 0,C 180,E1 -9624.037,E2 -9624.037} C_VEL
LIN {X 0,Y 425.578,Z 353.474,A -85,B 0,C 180,E1 -9628.106,E2 -9628.106} C_VEL
LIN {X 0,Y 425.705,Z 353.458,A -85,B 0,C 180,E1 -9629.999,E2 -9629.999} C_VEL
LIN {X 0,Y 425.559,Z 353.474,A -85,B 0,C 180,E1 -9632.839,E2 -9632.839} C_VEL
LIN {X 0,Y 425.533,Z 353.478,A -85,B 0,C 180,E1 -9636.638,E2 -9636.638} C_VEL
LIN {X 0,Y 425.402,Z 353.494,A -85,B 0,C 180,E1 -9639.508,E2 -9639.508} C_VEL
LIN {X 0,Y 425.393,Z 353.495,A -85,B 0,C 180,E1 -9642.903,E2 -9642.903} C_VEL
LIN {X 0,Y 425.369,Z 353.498,A -85,B 0,C 180,E1 -9646.608,E2 -9646.608} C_VEL
LIN {X 0,Y 425.327,Z 353.503,A -85,B 0,C 180,E1 -9649.635,E2 -9649.635} C_VEL
LIN {X 0,Y 425.305,Z 353.505,A -85,B 0,C 180,E1 -9653.364,E2 -9653.364} C_VEL
LIN {X 0,Y 425.346,Z 353.5,A -85,B 0,C 180,E1 -9656.843,E2 -9656.843} C_VEL
LIN {X 0,Y 425.315,Z 353.506,A -85,B 0,C 180,E1 -9659.716,E2 -9659.716} C_VEL
LIN {X 0,Y 425.28,Z 353.508,A -85,B 0,C 180,E1 -9663.047,E2 -9663.047} C_VEL
LIN {X 0,Y 425.28,Z 353.513,A -85,B 0,C 180,E1 -9665.928,E2 -9665.928} C_VEL
LIN {X 0,Y 425.31,Z 353.504,A -85,B 0,C 180,E1 -9669.045,E2 -9669.045} C_VEL
LIN {X 0,Y 425.325,Z 353.502,A -85,B 0,C 180,E1 -9672.645,E2 -9672.645} C_VEL
LIN {X 0,Y 425.327,Z 353.506,A -85,B 0,C 180,E1 -9676.053,E2 -9676.053} C_VEL
LIN {X 0,Y 425.303,Z 353.505,A -85,B 0,C 180,E1 -9678.625,E2 -9678.625} C_VEL
LIN {X 0,Y 425.318,Z 353.503,A -85,B 0,C 180,E1 -9681.104,E2 -9681.104} C_VEL
LIN {X 0,Y 425.292,Z 353.506,A -85,B 0,C 180,E1 -9684.663,E2 -9684.663} C_VEL
LIN {X 0,Y 425.258,Z 353.513,A -85,B 0,C 180,E1 -9688.073,E2 -9688.073} C_VEL
LIN {X 0,Y 425.329,Z 353.503,A -85,B 0,C 180,E1 -9691.368,E2 -9691.368} C_VEL
LIN {X 0,Y 425.286,Z 353.506,A -85,B 0,C 180,E1 -9694.554,E2 -9694.554} C_VEL
LIN {X 0,Y 425.278,Z 353.513,A -85,B 0,C 180,E1 -9697.661,E2 -9697.661} C_VEL
LIN {X 0,Y 425.352,Z 353.498,A -85,B 0,C 180,E1 -9700.704,E2 -9700.704} C_VEL
LIN {X 0,Y 425.389,Z 353.5,A -85,B 0,C 180,E1 -9703.688,E2 -9703.688} C_VEL
LIN {X 0,Y 425.42,Z 353.496,A -85,B 0,C 180,E1 -9707.599,E2 -9707.599} C_VEL
LIN {X 0,Y 425.433,Z 353.493,A -85,B 0,C 180,E1 -9711.45,E2 -9711.45} C_VEL
LIN {X 0,Y 425.545,Z 353.474,A -85,B 0,C 180,E1 -9714.313,E2 -9714.313} C_VEL
LIN {X 0,Y 425.566,Z 353.472,A -85,B 0,C 180,E1 -9718.107,E2 -9718.107} C_VEL
LIN {X 0,Y 425.695,Z 353.456,A -85,B 0,C 180,E1 -9720,E2 -9720} C_VEL
LIN {X 0,Y 425.549,Z 353.473,A -85,B 0,C 180,E1 -9722.84,E2 -9722.84} C_VEL
LIN {X 0,Y 425.569,Z 353.475,A -85,B 0,C 180,E1 -9725.687,E2 -9725.687} C_VEL
LIN {X 0,Y 425.433,Z 353.487,A -85,B 0,C 180,E1 -9728.55,E2 -9728.55} C_VEL
LIN {X 0,Y 425.422,Z 353.488,A -85,B 0,C 180,E1 -9732.402,E2 -9732.402} C_VEL
LIN {X 0,Y 425.379,Z 353.494,A -85,B 0,C 180,E1 -9736.312,E2 -9736.312} C_VEL
LIN {X 0,Y 425.319,Z 353.505,A -85,B 0,C 180,E1 -9739.636,E2 -9739.636} C_VEL
LIN {X 0,Y 425.298,Z 353.511,A -85,B 0,C 180,E1 -9743.366,E2 -9743.366} C_VEL
LIN {X 0,Y 425.34,Z 353.501,A -85,B 0,C 180,E1 -9746.845,E2 -9746.845} C_VEL
LIN {X 0,Y 425.283,Z 353.508,A -85,B 0,C 180,E1 -9749.72,E2 -9749.72} C_VEL
LIN {X 0,Y 425.275,Z 353.512,A -85,B 0,C 180,E1 -9753.049,E2 -9753.049} C_VEL
LIN {X 0,Y 425.278,Z 353.508,A -85,B 0,C 180,E1 -9755.93,E2 -9755.93} C_VEL
LIN {X 0,Y 425.307,Z 353.509,A -85,B 0,C 180,E1 -9759.047,E2 -9759.047} C_VEL
LIN {X 0,Y 425.326,Z 353.503,A -85,B 0,C 180,E1 -9762.647,E2 -9762.647} C_VEL
LIN {X 0,Y 425.313,Z 353.503,A -85,B 0,C 180,E1 -9766.053,E2 -9766.053} C_VEL
LIN {X 0,Y 425.305,Z 353.506,A -85,B 0,C 180,E1 -9768.627,E2 -9768.627} C_VEL
LIN {X 0,Y 425.321,Z 353.508,A -85,B 0,C 180,E1 -9771.106,E2 -9771.106} C_VEL
LIN {X 0,Y 425.297,Z 353.507,A -85,B 0,C 180,E1 -9774.666,E2 -9774.666} C_VEL
LIN {X 0,Y 425.272,Z 353.509,A -85,B 0,C 180,E1 -9778.075,E2 -9778.075} C_VEL
LIN {X 0,Y 425.397,Z 353.562,A -85,B 0,C 180,E1 -9780.669,E2 -9780.669} C_VEL
LIN {X 0,Y 428.744,Z 369.606,A -85,B 0,C 180,E1 -9783.732,E2 -9783.732} C_VEL
LIN {X 0,Y 428.847,Z 373.648,A -85,B 0,C 180,E1 -9784.455,E2 -9784.455} C_VEL
LIN {X 0,Y 427.539,Z 394.423,A -85,B 0,C 180,E1 -9788.041,E2 -9788.041} C_VEL
LIN {X 0,Y 426.455,Z 414.782,A -85,B 0,C 180,E1 -9791.505,E2 -9791.505} C_VEL
LIN {X 0,Y 429.777,Z 441.56,A -85,B 0,C 180,E1 -9792.182,E2 -9792.182} C_VEL
LIN {X 0,Y 428.497,Z 524.207,A -85,B 0,C 180,E1 -9793.842,E2 -9793.842} C_VEL
LIN {X 0,Y 427.95,Z 538.082,A -85,B 0,C 180,E1 -9794.31,E2 -9794.31} C_VEL
LIN {X 0,Y 427.361,Z 550.66,A -85,B 0,C 180,E1 -9794.929,E2 -9794.929} C_VEL
LIN {X 0,Y 426.765,Z 562.357,A -85,B 0,C 180,E1 -9795.7,E2 -9795.7} C_VEL
LIN {X 0,Y 426.056,Z 574.443,A -85,B 0,C 180,E1 -9796.715,E2 -9796.715} C_VEL
LIN {X 0,Y 425.601,Z 584.058,A -85,B 0,C 180,E1 -9797.726,E2 -9797.726} C_VEL
LIN {X 0,Y 425.21,Z 592.527,A -85,B 0,C 180,E1 -9798.803,E2 -9798.803} C_VEL
LIN {X 0,Y 424.76,Z 601.729,A -85,B 0,C 180,E1 -9800.237,E2 -9800.237} C_VEL
LIN {X 0,Y 424.5,Z 609.128,A -85,B 0,C 180,E1 -9801.672,E2 -9801.672} C_VEL
LIN {X 0,Y 424.35,Z 614.099,A -85,B 0,C 180,E1 -9802.866,E2 -9802.866} C_VEL
LIN {X 0,Y 424.302,Z 618.899,A -85,B 0,C 180,E1 -9804.298,E2 -9804.298} C_VEL
LIN {X 0,Y 424.219,Z 622.504,A -85,B 0,C 180,E1 -9805.726,E2 -9805.726} C_VEL
LIN {X 0,Y 424.312,Z 625.038,A -85,B 0,C 180,E1 -9807.153,E2 -9807.153} C_VEL
LIN {X 0,Y 424.349,Z 626.157,A -85,B 0,C 180,E1 -9808.103,E2 -9808.103} C_VEL
LIN {X 0,Y 424.264,Z 626.812,A -85,B 0,C 180,E1 -9809.052,E2 -9809.052} C_VEL
LIN {X 0,Y 424.242,Z 627.055,A -85,B 0,C 180,E1 -9810.001,E2 -9810.001} C_VEL
LIN {X 0,Y 424.265,Z 626.876,A -85,B 0,C 180,E1 -9810.95,E2 -9810.95} C_VEL
LIN {X 0,Y 424.307,Z 626.226,A -85,B 0,C 180,E1 -9811.899,E2 -9811.899} C_VEL
LIN {X 0,Y 424.329,Z 625.148,A -85,B 0,C 180,E1 -9812.849,E2 -9812.849} C_VEL
LIN {X 0,Y 424.266,Z 623.636,A -85,B 0,C 180,E1 -9813.8,E2 -9813.8} C_VEL
LIN {X 0,Y 424.281,Z 620.484,A -85,B 0,C 180,E1 -9815.228,E2 -9815.228} C_VEL
LIN {X 0,Y 424.358,Z 616.23,A -85,B 0,C 180,E1 -9816.658,E2 -9816.658} C_VEL
LIN {X 0,Y 424.495,Z 609.704,A -85,B 0,C 180,E1 -9818.331,E2 -9818.331} C_VEL
LIN {X 0,Y 424.745,Z 602.581,A -85,B 0,C 180,E1 -9819.766,E2 -9819.766} C_VEL
LIN {X 0,Y 425.222,Z 593.78,A -85,B 0,C 180,E1 -9821.199,E2 -9821.199} C_VEL
LIN {X 0,Y 425.686,Z 584.748,A -85,B 0,C 180,E1 -9822.395,E2 -9822.395} C_VEL
LIN {X 0,Y 426.329,Z 573.93,A -85,B 0,C 180,E1 -9823.563,E2 -9823.563} C_VEL
LIN {X 0,Y 427.078,Z 562.777,A -85,B 0,C 180,E1 -9824.535,E2 -9824.535} C_VEL
LIN {X 0,Y 427.8,Z 550.744,A -85,B 0,C 180,E1 -9825.362,E2 -9825.362} C_VEL
LIN {X 0,Y 428.519,Z 537.252,A -85,B 0,C 180,E1 -9826.068,E2 -9826.068} C_VEL
LIN {X 0,Y 429.27,Z 523.5,A -85,B 0,C 180,E1 -9826.558,E2 -9826.558} C_VEL
LIN {X 0,Y 429.837,Z 493.063,A -85,B 0,C 180,E1 -9827.23,E2 -9827.23} C_VEL
LIN {X 0,Y 431.016,Z 441.341,A -85,B 0,C 180,E1 -9828.356,E2 -9828.356} C_VEL
LIN {X 0,Y 428.471,Z 420.013,A -85,B 0,C 180,E1 -9829.02,E2 -9829.02} C_VEL
LIN {X 0,Y 426.764,Z 409.909,A -85,B 0,C 180,E1 -9829.387,E2 -9829.387} C_VEL
LIN {X 0,Y 428.112,Z 389.581,A -85,B 0,C 180,E1 -9833.025,E2 -9833.025} C_VEL
LIN {X 0,Y 429.517,Z 372.483,A -85,B 0,C 180,E1 -9836.219,E2 -9836.219} C_VEL
LIN {X 0,Y 427.832,Z 363.409,A -85,B 0,C 180,E1 -9838.203,E2 -9838.203} C_VEL
LIN {X 0,Y 425.312,Z 353.509,A -85,B 0,C 180,E1 -9840.634,E2 -9840.634} C_VEL
LIN {X 0,Y 425.317,Z 353.508,A -85,B 0,C 180,E1 -9844.289,E2 -9844.289} C_VEL
LIN {X 0,Y 425.285,Z 353.511,A -85,B 0,C 180,E1 -9847.695,E2 -9847.695} C_VEL
LIN {X 0,Y 425.287,Z 353.511,A -85,B 0,C 180,E1 -9850.521,E2 -9850.521} C_VEL
LIN {X 0,Y 425.263,Z 353.512,A -85,B 0,C 180,E1 -9853.351,E2 -9853.351} C_VEL
LIN {X 0,Y 425.263,Z 353.512,A -85,B 0,C 180,E1 -9856.649,E2 -9856.649} C_VEL
LIN {X 0,Y 425.295,Z 353.508,A -85,B 0,C 180,E1 -9859.873,E2 -9859.873} C_VEL
LIN {X 0,Y 425.284,Z 353.51,A -85,B 0,C 180,E1 -9862.489,E2 -9862.489} C_VEL
LIN {X 0,Y 425.313,Z 353.505,A -85,B 0,C 180,E1 -9865.818,E2 -9865.818} C_VEL
LIN {X 0,Y 425.296,Z 353.509,A -85,B 0,C 180,E1 -9869.239,E2 -9869.239} C_VEL
LIN {X 0,Y 425.354,Z 353.503,A -85,B 0,C 180,E1 -9872.443,E2 -9872.443} C_VEL
LIN {X 0,Y 425.357,Z 353.502,A -85,B 0,C 180,E1 -9875.602,E2 -9875.602} C_VEL
LIN {X 0,Y 425.31,Z 353.523,A -85,B 0,C 180,E1 -9878.936,E2 -9878.936} C_VEL
LIN {X 0,Y 426.527,Z 358.793,A -85,B 0,C 180,E1 -9880.703,E2 -9880.703} C_VEL
LIN {X 0,Y 431.967,Z 371.565,A -85,B 0,C 180,E1 -9881.392,E2 -9881.392} C_VEL
LIN {X 0,Y 432.123,Z 373.467,A -85,B 0,C 180,E1 -9881.449,E2 -9881.449} C_VEL
LIN {X 0,Y 430.029,Z 453.987,A -85,B 0,C 180,E1 -9883.228,E2 -9883.228} C_VEL
LIN {X 0,Y 429.765,Z 468.696,A -85,B 0,C 180,E1 -9883.615,E2 -9883.615} C_VEL
LIN {X 0,Y 429.357,Z 481.544,A -85,B 0,C 180,E1 -9884.148,E2 -9884.148} C_VEL
LIN {X 0,Y 428.891,Z 493.071,A -85,B 0,C 180,E1 -9884.8,E2 -9884.8} C_VEL
LIN {X 0,Y 428.373,Z 504.411,A -85,B 0,C 180,E1 -9885.632,E2 -9885.632} C_VEL
LIN {X 0,Y 427.592,Z 515.922,A -85,B 0,C 180,E1 -9886.696,E2 -9886.696} C_VEL
LIN {X 0,Y 426.936,Z 526.141,A -85,B 0,C 180,E1 -9887.884,E2 -9887.884} C_VEL
LIN {X 0,Y 426.37,Z 535.878,A -85,B 0,C 180,E1 -9889.313,E2 -9889.313} C_VEL
LIN {X 0,Y 425.825,Z 543.695,A -85,B 0,C 180,E1 -9890.74,E2 -9890.74} C_VEL
LIN {X 0,Y 425.431,Z 548.97,A -85,B 0,C 180,E1 -9891.928,E2 -9891.928} C_VEL
LIN {X 0,Y 424.944,Z 554.08,A -85,B 0,C 180,E1 -9893.352,E2 -9893.352} C_VEL
LIN {X 0,Y 424.875,Z 557.971,A -85,B 0,C 180,E1 -9894.78,E2 -9894.78} C_VEL
LIN {X 0,Y 424.759,Z 560.806,A -85,B 0,C 180,E1 -9896.205,E2 -9896.205} C_VEL
LIN {X 0,Y 424.565,Z 562.127,A -85,B 0,C 180,E1 -9897.153,E2 -9897.153} C_VEL
LIN {X 0,Y 424.384,Z 563.038,A -85,B 0,C 180,E1 -9898.102,E2 -9898.102} C_VEL
LIN {X 0,Y 424.286,Z 563.54,A -85,B 0,C 180,E1 -9899.051,E2 -9899.051} C_VEL
LIN {X 0,Y 424.259,Z 563.583,A -85,B 0,C 180,E1 -9900,E2 -9900} C_VEL
LIN {X 0,Y 424.284,Z 563.202,A -85,B 0,C 180,E1 -9900.949,E2 -9900.949} C_VEL
LIN {X 0,Y 424.378,Z 562.418,A -85,B 0,C 180,E1 -9901.898,E2 -9901.898} C_VEL
LIN {X 0,Y 424.471,Z 561.215,A -85,B 0,C 180,E1 -9902.847,E2 -9902.847} C_VEL
LIN {X 0,Y 424.612,Z 558.571,A -85,B 0,C 180,E1 -9904.271,E2 -9904.271} C_VEL
LIN {X 0,Y 424.631,Z 554.888,A -85,B 0,C 180,E1 -9905.699,E2 -9905.699} C_VEL
LIN {X 0,Y 424.943,Z 550.133,A -85,B 0,C 180,E1 -9907.1,E2 -9907.1} C_VEL
LIN {X 0,Y 425.179,Z 543.884,A -85,B 0,C 180,E1 -9908.555,E2 -9908.555} C_VEL
LIN {X 0,Y 425.603,Z 536.211,A -85,B 0,C 180,E1 -9909.985,E2 -9909.985} C_VEL
LIN {X 0,Y 426.036,Z 528.381,A -85,B 0,C 180,E1 -9911.176,E2 -9911.176} C_VEL
LIN {X 0,Y 426.543,Z 518.849,A -85,B 0,C 180,E1 -9912.368,E2 -9912.368} C_VEL
LIN {X 0,Y 427.155,Z 508.021,A -85,B 0,C 180,E1 -9913.459,E2 -9913.459} C_VEL
LIN {X 0,Y 427.538,Z 496.494,A -85,B 0,C 180,E1 -9914.396,E2 -9914.396} C_VEL
LIN {X 0,Y 428.007,Z 484.081,A -85,B 0,C 180,E1 -9915.171,E2 -9915.171} C_VEL
LIN {X 0,Y 428.521,Z 470.525,A -85,B 0,C 180,E1 -9915.792,E2 -9915.792} C_VEL
LIN {X 0,Y 428.797,Z 457.922,A -85,B 0,C 180,E1 -9916.178,E2 -9916.178} C_VEL
LIN {X 0,Y 430.076,Z 369.096,A -85,B 0,C 180,E1 -9917.953,E2 -9917.953} C_VEL
LIN {X 0,Y 425.379,Z 353.498,A -85,B 0,C 180,E1 -9918.482,E2 -9918.482} C_VEL
LIN {X 0,Y 425.297,Z 353.508,A -85,B 0,C 180,E1 -9922.27,E2 -9922.27} C_VEL
LIN {X 0,Y 425.328,Z 353.505,A -85,B 0,C 180,E1 -9924.658,E2 -9924.658} C_VEL
LIN {X 0,Y 425.353,Z 353.501,A -85,B 0,C 180,E1 -9927.557,E2 -9927.557} C_VEL
LIN {X 0,Y 425.293,Z 353.51,A -85,B 0,C 180,E1 -9930.816,E2 -9930.816} C_VEL
LIN {X 0,Y 425.316,Z 353.505,A -85,B 0,C 180,E1 -9934.287,E2 -9934.287} C_VEL
LIN {X 0,Y 425.283,Z 353.511,A -85,B 0,C 180,E1 -9937.694,E2 -9937.694} C_VEL
LIN {X 0,Y 425.286,Z 353.51,A -85,B 0,C 180,E1 -9940.52,E2 -9940.52} C_VEL
LIN {X 0,Y 425.262,Z 353.512,A -85,B 0,C 180,E1 -9943.35,E2 -9943.35} C_VEL
LIN {X 0,Y 425.262,Z 353.515,A -85,B 0,C 180,E1 -9946.648,E2 -9946.648} C_VEL
LIN {X 0,Y 425.294,Z 353.508,A -85,B 0,C 180,E1 -9949.873,E2 -9949.873} C_VEL
LIN {X 0,Y 425.282,Z 353.511,A -85,B 0,C 180,E1 -9952.488,E2 -9952.488} C_VEL
LIN {X 0,Y 425.312,Z 353.506,A -85,B 0,C 180,E1 -9955.817,E2 -9955.817} C_VEL
LIN {X 0,Y 425.294,Z 353.508,A -85,B 0,C 180,E1 -9959.238,E2 -9959.238} C_VEL
LIN {X 0,Y 425.353,Z 353.503,A -85,B 0,C 180,E1 -9962.442,E2 -9962.442} C_VEL
LIN {X 0,Y 425.355,Z 353.5,A -85,B 0,C 180,E1 -9965.601,E2 -9965.601} C_VEL
LIN {X 0,Y 425.297,Z 353.509,A -85,B 0,C 180,E1 -9968.681,E2 -9968.681} C_VEL
LIN {X 0,Y 425.337,Z 353.502,A -85,B 0,C 180,E1 -9971.702,E2 -9971.702} C_VEL
LIN {X 0,Y 425.352,Z 353.502,A -85,B 0,C 180,E1 -9974.67,E2 -9974.67} C_VEL
LIN {X 0,Y 425.415,Z 353.492,A -85,B 0,C 180,E1 -9977.597,E2 -9977.597} C_VEL
LIN {X 0,Y 425.445,Z 353.489,A -85,B 0,C 180,E1 -9981.449,E2 -9981.449} C_VEL
LIN {X 0,Y 425.533,Z 353.479,A -85,B 0,C 180,E1 -9984.037,E2 -9984.037} C_VEL
LIN {X 0,Y 424.915,Z 353.561,A -85,B 0,C 180,E1 -9984.825,E2 -9984.825} C_VEL
LIN {X 0,Y 422.118,Z 353.913,A -85,B 0,C 180,E1 -9986.108,E2 -9986.108} C_VEL
LIN {X 0,Y 419.705,Z 354.211,A -85,B 0,C 180,E1 -9987.142,E2 -9987.142} C_VEL
LIN {X 0,Y 418.637,Z 354.34,A -85,B 0,C 180,E1 -9987.942,E2 -9987.942} C_VEL
LIN {X 0,Y 418.534,Z 354.35,A -85,B 0,C 180,E1 -9988.213,E2 -9988.213} C_VEL
LIN {X 0,Y 418.675,Z 354.334,A -85,B 0,C 180,E1 -9989.999,E2 -9989.999} C_VEL
LIN {X 0,Y 418.512,Z 354.352,A -85,B 0,C 180,E1 -9992.887,E2 -9992.887} C_VEL
LIN {X 0,Y 418.495,Z 354.354,A -85,B 0,C 180,E1 -9996.75,E2 -9996.75} C_VEL
LIN {X 0,Y 418.342,Z 354.374,A -85,B 0,C 180,E1 -9999.67,E2 -9999.67} C_VEL
LIN {X 0,Y 418.346,Z 354.372,A -85,B 0,C 180,E1 -10003,E2 -10003} C_VEL
LIN {X 0,Y 418.319,Z 354.376,A -85,B 0,C 180,E1 -10006.738,E2 -10006.738} C_VEL
LIN {X 0,Y 418.269,Z 354.384,A -85,B 0,C 180,E1 -10009.789,E2 -10009.789} C_VEL
LIN {X 0,Y 418.236,Z 354.386,A -85,B 0,C 180,E1 -10012.735,E2 -10012.735} C_VEL
LIN {X 0,Y 418.268,Z 354.385,A -85,B 0,C 180,E1 -10015.903,E2 -10015.903} C_VEL
LIN {X 0,Y 418.271,Z 354.382,A -85,B 0,C 180,E1 -10019.16,E2 -10019.16} C_VEL
LIN {X 0,Y 418.256,Z 354.383,A -85,B 0,C 180,E1 -10022.843,E2 -10022.843} C_VEL
LIN {X 0,Y 418.244,Z 354.387,A -85,B 0,C 180,E1 -10026.238,E2 -10026.238} C_VEL
LIN {X 0,Y 418.262,Z 354.385,A -85,B 0,C 180,E1 -10029.679,E2 -10029.679} C_VEL
LIN {X 0,Y 418.279,Z 354.381,A -85,B 0,C 180,E1 -10032.329,E2 -10032.329} C_VEL
LIN {X 0,Y 418.268,Z 354.382,A -85,B 0,C 180,E1 -10035.113,E2 -10035.113} C_VEL
LIN {X 0,Y 418.286,Z 354.384,A -85,B 0,C 180,E1 -10037.772,E2 -10037.772} C_VEL
LIN {X 0,Y 418.26,Z 354.385,A -85,B 0,C 180,E1 -10041.559,E2 -10041.559} C_VEL
LIN {X 0,Y 418.252,Z 354.384,A -85,B 0,C 180,E1 -10045.158,E2 -10045.158} C_VEL
LIN {X 0,Y 418.237,Z 354.387,A -85,B 0,C 180,E1 -10047.471,E2 -10047.471} C_VEL
LIN {X 0,Y 418.268,Z 354.381,A -85,B 0,C 180,E1 -10050.893,E2 -10050.893} C_VEL
LIN {X 0,Y 418.262,Z 354.384,A -85,B 0,C 180,E1 -10054.095,E2 -10054.095} C_VEL
LIN {X 0,Y 418.229,Z 354.387,A -85,B 0,C 180,E1 -10057.263,E2 -10057.263} C_VEL
LIN {X 0,Y 418.274,Z 354.38,A -85,B 0,C 180,E1 -10060.364,E2 -10060.364} C_VEL
LIN {X 0,Y 418.316,Z 354.378,A -85,B 0,C 180,E1 -10063.405,E2 -10063.405} C_VEL
LIN {X 0,Y 418.345,Z 354.371,A -85,B 0,C 180,E1 -10066.993,E2 -10066.993} C_VEL
LIN {X 0,Y 418.351,Z 354.37,A -85,B 0,C 180,E1 -10070.329,E2 -10070.329} C_VEL
LIN {X 0,Y 418.484,Z 354.356,A -85,B 0,C 180,E1 -10073.249,E2 -10073.249} C_VEL
LIN {X 0,Y 418.333,Z 354.375,A -85,B 0,C 180,E1 -10075.182,E2 -10075.182} C_VEL
LIN {X 0,Y 418.535,Z 354.348,A -85,B 0,C 180,E1 -10078.076,E2 -10078.076} C_VEL
LIN {X 0,Y 418.665,Z 354.332,A -85,B 0,C 180,E1 -10080,E2 -10080} C_VEL
LIN {X 0,Y 418.503,Z 354.351,A -85,B 0,C 180,E1 -10082.888,E2 -10082.888} C_VEL
LIN {X 0,Y 418.524,Z 354.351,A -85,B 0,C 180,E1 -10085.783,E2 -10085.783} C_VEL
LIN {X 0,Y 418.391,Z 354.365,A -85,B 0,C 180,E1 -10088.695,E2 -10088.695} C_VEL
LIN {X 0,Y 418.326,Z 354.377,A -85,B 0,C 180,E1 -10091.631,E2 -10091.631} C_VEL
LIN {X 0,Y 418.298,Z 354.376,A -85,B 0,C 180,E1 -10094.597,E2 -10094.597} C_VEL
LIN {X 0,Y 418.279,Z 354.383,A -85,B 0,C 180,E1 -10097.604,E2 -10097.604} C_VEL
LIN {X 0,Y 418.241,Z 354.384,A -85,B 0,C 180,E1 -10100.664,E2 -10100.664} C_VEL
LIN {X 0,Y 418.279,Z 354.381,A -85,B 0,C 180,E1 -10103.782,E2 -10103.782} C_VEL
LIN {X 0,Y 418.301,Z 354.38,A -85,B 0,C 180,E1 -10107.071,E2 -10107.071} C_VEL
LIN {X 0,Y 418.236,Z 354.384,A -85,B 0,C 180,E1 -10110.273,E2 -10110.273} C_VEL
LIN {X 0,Y 418.241,Z 354.386,A -85,B 0,C 180,E1 -10113.678,E2 -10113.678} C_VEL
LIN {X 0,Y 418.241,Z 354.39,A -85,B 0,C 180,E1 -10117.224,E2 -10117.224} C_VEL
LIN {X 0,Y 418.26,Z 354.383,A -85,B 0,C 180,E1 -10119.681,E2 -10119.681} C_VEL
LIN {X 0,Y 418.279,Z 354.379,A -85,B 0,C 180,E1 -10122.331,E2 -10122.331} C_VEL
LIN {X 0,Y 418.269,Z 354.387,A -85,B 0,C 180,E1 -10125.115,E2 -10125.115} C_VEL
LIN {X 0,Y 418.288,Z 354.379,A -85,B 0,C 180,E1 -10127.775,E2 -10127.775} C_VEL
LIN {X 0,Y 418.263,Z 354.383,A -85,B 0,C 180,E1 -10131.561,E2 -10131.561} C_VEL
LIN {X 0,Y 418.256,Z 354.387,A -85,B 0,C 180,E1 -10135.16,E2 -10135.16} C_VEL
LIN {X 0,Y 418.247,Z 354.385,A -85,B 0,C 180,E1 -10137.474,E2 -10137.474} C_VEL
LIN {X 0,Y 418.352,Z 354.548,A -85,B 0,C 180,E1 -10140.467,E2 -10140.467} C_VEL
LIN {X 0,Y 421.867,Z 371.41,A -85,B 0,C 180,E1 -10143.736,E2 -10143.736} C_VEL
LIN {X 0,Y 421.672,Z 377.647,A -85,B 0,C 180,E1 -10144.85,E2 -10144.85} C_VEL
LIN {X 0,Y 420.536,Z 395.096,A -85,B 0,C 180,E1 -10147.914,E2 -10147.914} C_VEL
LIN {X 0,Y 419.449,Z 414.432,A -85,B 0,C 180,E1 -10151.248,E2 -10151.248} C_VEL
LIN {X 0,Y 422.856,Z 442.939,A -85,B 0,C 180,E1 -10151.978,E2 -10151.978} C_VEL
LIN {X 0,Y 421.531,Z 524.205,A -85,B 0,C 180,E1 -10153.661,E2 -10153.661} C_VEL
LIN {X 0,Y 420.983,Z 537.889,A -85,B 0,C 180,E1 -10154.136,E2 -10154.136} C_VEL
LIN {X 0,Y 420.428,Z 549.862,A -85,B 0,C 180,E1 -10154.736,E2 -10154.736} C_VEL
LIN {X 0,Y 419.746,Z 562.4,A -85,B 0,C 180,E1 -10155.579,E2 -10155.579} C_VEL
LIN {X 0,Y 419.026,Z 574.303,A -85,B 0,C 180,E1 -10156.604,E2 -10156.604} C_VEL
LIN {X 0,Y 418.547,Z 583.899,A -85,B 0,C 180,E1 -10157.639,E2 -10157.639} C_VEL
LIN {X 0,Y 418.111,Z 593.152,A -85,B 0,C 180,E1 -10158.856,E2 -10158.856} C_VEL
LIN {X 0,Y 417.653,Z 602.172,A -85,B 0,C 180,E1 -10160.314,E2 -10160.314} C_VEL
LIN {X 0,Y 417.413,Z 609.347,A -85,B 0,C 180,E1 -10161.773,E2 -10161.773} C_VEL
LIN {X 0,Y 417.254,Z 615.055,A -85,B 0,C 180,E1 -10163.23,E2 -10163.23} C_VEL
LIN {X 0,Y 417.242,Z 619.501,A -85,B 0,C 180,E1 -10164.686,E2 -10164.686} C_VEL
LIN {X 0,Y 417.175,Z 622.787,A -85,B 0,C 180,E1 -10166.137,E2 -10166.137} C_VEL
